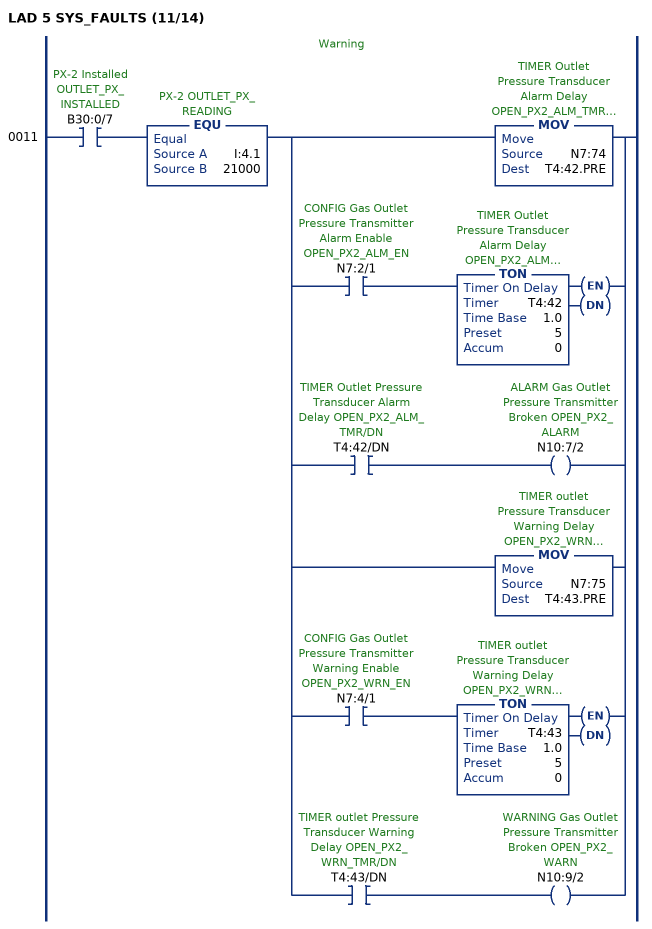
% Rung: 11 %
% Warning %
SOR XIC B30:0/7 EQU I:4.1 21000 BST MOV N7:74 T4:42.PRE NXB XIC N7:2/1 TON T4:42 1.0 5 0 NXB XIC T4:42/DN OTE N10:7/2 NXB MOV N7:75 T4:43.PRE NXB XIC N7:4/1 TON T4:43 1.0 5 0 NXB XIC T4:43/DN OTE N10:9/2 BND EOR
%   B30:0/7  OUTLET_PX_INSTALLED  "PX-2 Installed" %
%   I:4.1  OUTLET_PX_READING  "PX-2" %
%   N7:74  OPEN_PX2_ALM_DLY  "CONFIG Gas Outlet Pressure Transducer Alarm Delay" %
%   T4:42  OPEN_PX2_ALM_TMR  "TIMER Outlet Pressure Transducer Alarm Delay" %
%   N7:2/1  OPEN_PX2_ALM_EN  "CONFIG Gas Outlet Pressure Transmitter Alarm Enable" %
%   N10:7/2  OPEN_PX2_ALARM  "ALARM Gas Outlet Pressure Transmitter Broken" %
%   N7:75  OPEN_PX2_WRN_DLY  "CONFIG Gas Outlet Pressure Transducer Warning Delay" %
%   T4:43  OPEN_PX2_WRN_TMR  "TIMER outlet Pressure Transducer Warning Delay" %
%   N7:4/1  OPEN_PX2_WRN_EN  "CONFIG Gas Outlet Pressure Transmitter Warning Enable" %
%   N10:9/2  OPEN_PX2_WARN  "WARNING Gas Outlet Pressure Transmitter Broken" %

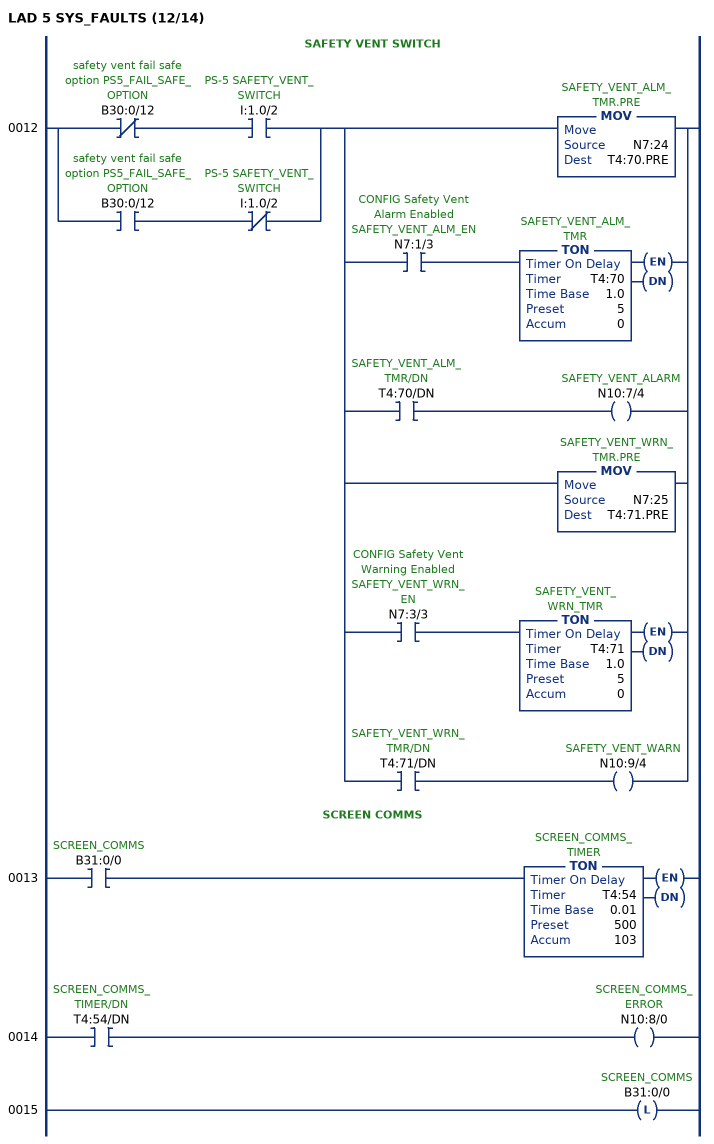
% Rung: 12 %
% TITLE: SAFETY VENT SWITCH %
SOR BST XIO B30:0/12 XIC I:1.0/2 NXB XIC B30:0/12 XIO I:1.0/2 BND BST MOV N7:24 T4:70.PRE NXB XIC N7:1/3 TON T4:70 1.0 5 0 NXB XIC T4:70/DN OTE N10:7/4 NXB MOV N7:25 T4:71.PRE NXB XIC N7:3/3 TON T4:71 1.0 5 0 NXB XIC T4:71/DN OTE N10:9/4 BND EOR
%   B30:0/12  PS5_FAIL_SAFE_OPTION  "safety vent fail safe option" %
%   I:1.0/2  SAFETY_VENT_SWITCH  "PS-5" %
%   N7:24  SAFETY_VENT_ALM_DLY  "CONFIG Safety Vent Alarm Delay" %
%   T4:70  SAFETY_VENT_ALM_TMR %
%   N7:1/3  SAFETY_VENT_ALM_EN  "CONFIG Safety Vent Alarm Enabled" %
%   N10:7/4  SAFETY_VENT_ALARM %
%   N7:25  SAFETY_VENT_WRN_DLY  "CONFIG Safety Vent Warning Delay" %
%   T4:71  SAFETY_VENT_WRN_TMR %
%   N7:3/3  SAFETY_VENT_WRN_EN  "CONFIG Safety Vent Warning Enabled" %
%   N10:9/4  SAFETY_VENT_WARN %
% Rung: 13 %
% TITLE: SCREEN COMMS %
SOR XIC B31:0/0 TON T4:54 0.01 500 103 EOR
%   B31:0/0  SCREEN_COMMS %
%   T4:54  SCREEN_COMMS_TIMER %
% Rung: 14 %
SOR XIC T4:54/DN OTE N10:8/0 EOR
%   T4:54  SCREEN_COMMS_TIMER %
%   N10:8/0  SCREEN_COMMS_ERROR %
% Rung: 15 %
SOR OTL B31:0/0 EOR
%   B31:0/0  SCREEN_COMMS %

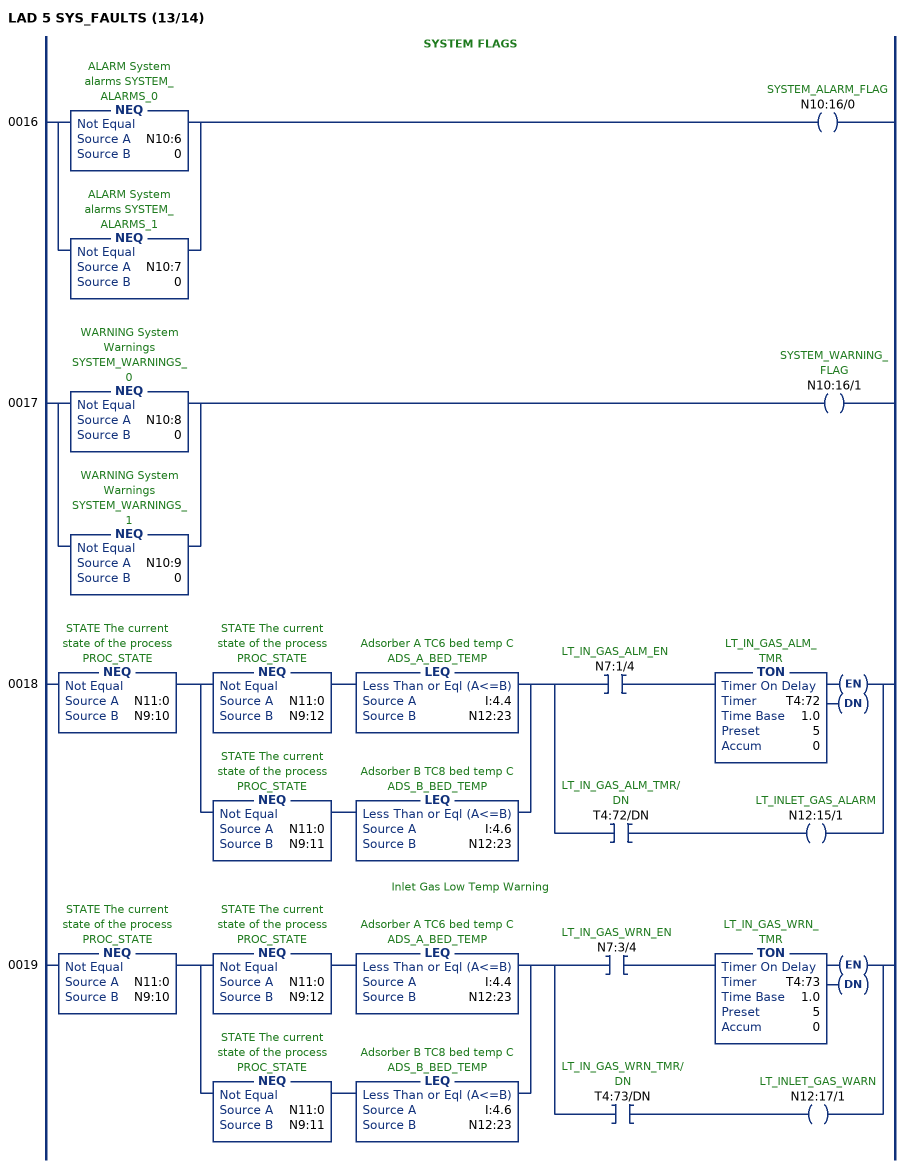
% Rung: 16 %
% TITLE: SYSTEM FLAGS %
SOR BST NEQ N10:6 0 NXB NEQ N10:7 0 BND OTE N10:16/0 EOR
%   N10:6  SYSTEM_ALARMS_0  "ALARM System alarms" %
%   N10:7  SYSTEM_ALARMS_1  "ALARM System alarms" %
%   N10:16/0  SYSTEM_ALARM_FLAG %
% Rung: 17 %
SOR BST NEQ N10:8 0 NXB NEQ N10:9 0 BND OTE N10:16/1 EOR
%   N10:8  SYSTEM_WARNINGS_0  "WARNING System Warnings" %
%   N10:9  SYSTEM_WARNINGS_1  "WARNING System Warnings" %
%   N10:16/1  SYSTEM_WARNING_FLAG %
% Rung: 18 %
SOR NEQ N11:0 N9:10 BST NEQ N11:0 N9:12 LEQ I:4.4 N12:23 NXB NEQ N11:0 N9:11 LEQ I:4.6 N12:23 BND BST XIC N7:1/4 TON T4:72 1.0 5 0 NXB XIC T4:72/DN OTE N12:15/1 BND EOR
%   N11:0  PROC_STATE  "STATE The current state of the process" %
%   N9:10  PROCESS_STANDBY %
%   N9:12  PROC_REGEN_A  "STATE Process Purify B" %
%   I:4.4  ADS_A_BED_TEMP  "Adsorber A TC6 bed temp C" %
%   N12:23  LT_INLET_GAS_ALM_SP %
%   N9:11  PROC_REGEN_B  "STATE Process Purify A" %
%   I:4.6  ADS_B_BED_TEMP  "Adsorber B TC8 bed temp C" %
%   N7:1/4  LT_IN_GAS_ALM_EN %
%   T4:72  LT_IN_GAS_ALM_TMR %
%   N12:15/1  LT_INLET_GAS_ALARM %
% Rung: 19 %
% Inlet Gas Low Temp Warning %
SOR NEQ N11:0 N9:10 BST NEQ N11:0 N9:12 LEQ I:4.4 N12:23 NXB NEQ N11:0 N9:11 LEQ I:4.6 N12:23 BND BST XIC N7:3/4 TON T4:73 1.0 5 0 NXB XIC T4:73/DN OTE N12:17/1 BND EOR
%   N11:0  PROC_STATE  "STATE The current state of the process" %
%   N9:10  PROCESS_STANDBY %
%   N9:12  PROC_REGEN_A  "STATE Process Purify B" %
%   I:4.4  ADS_A_BED_TEMP  "Adsorber A TC6 bed temp C" %
%   N12:23  LT_INLET_GAS_ALM_SP %
%   N9:11  PROC_REGEN_B  "STATE Process Purify A" %
%   I:4.6  ADS_B_BED_TEMP  "Adsorber B TC8 bed temp C" %
%   N7:3/4  LT_IN_GAS_WRN_EN %
%   T4:73  LT_IN_GAS_WRN_TMR %
%   N12:17/1  LT_INLET_GAS_WARN %

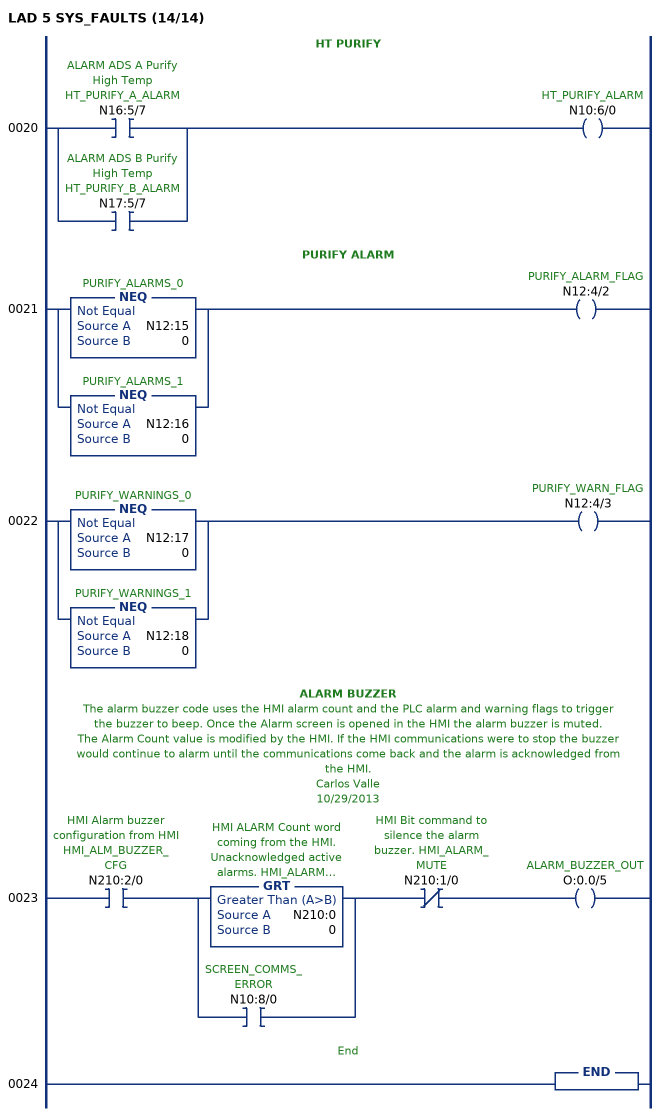
% Rung: 20 %
% TITLE: HT PURIFY %
SOR BST XIC N16:5/7 NXB XIC N17:5/7 BND OTE N10:6/0 EOR
%   N16:5/7  HT_PURIFY_A_ALARM  "ALARM ADS A Purify High Temp" %
%   N17:5/7  HT_PURIFY_B_ALARM  "ALARM ADS B Purify High Temp" %
%   N10:6/0  HT_PURIFY_ALARM %
% Rung: 21 %
% TITLE: PURIFY ALARM %
SOR BST NEQ N12:15 0 NXB NEQ N12:16 0 BND OTE N12:4/2 EOR
%   N12:15  PURIFY_ALARMS_0 %
%   N12:16  PURIFY_ALARMS_1 %
%   N12:4/2  PURIFY_ALARM_FLAG %
% Rung: 22 %
SOR BST NEQ N12:17 0 NXB NEQ N12:18 0 BND OTE N12:4/3 EOR
%   N12:17  PURIFY_WARNINGS_0 %
%   N12:18  PURIFY_WARNINGS_1 %
%   N12:4/3  PURIFY_WARN_FLAG %
% Rung: 23 %
% TITLE: ALARM BUZZER %
% The alarm buzzer code uses the HMI alarm count and the PLC alarm and warning flags to trigger the buzzer to beep. Once the Alarm screen is opened in the HMI the alarm buzzer is muted.
% The Alarm Count value is modified by the HMI. If the HMI communications were to stop the buzzer would continue to alarm until the communications come back and the alarm is acknowledged from the HMI.
% Carlos Valle
% 10/29/2013 %
SOR XIC N210:2/0 BST GRT N210:0 0 NXB XIC N10:8/0 BND XIO N210:1/0 OTE O:0.0/5 EOR
%   N210:2/0  HMI_ALM_BUZZER_CFG  "HMI Alarm buzzer configuration from HMI" %
%   N210:0  HMI_ALARM_COUNT  "HMI ALARM Count word coming from the HMI. Unacknowledged active alarms." %
%   N10:8/0  SCREEN_COMMS_ERROR %
%   N210:1/0  HMI_ALARM_MUTE  "HMI Bit command to silence the alarm buzzer." %
%   O:0.0/5  ALARM_BUZZER_OUT %
% Rung: 24 %
% End %
SOR END EOR

LADDER 6 "SYSTEM"    % Controls the system %
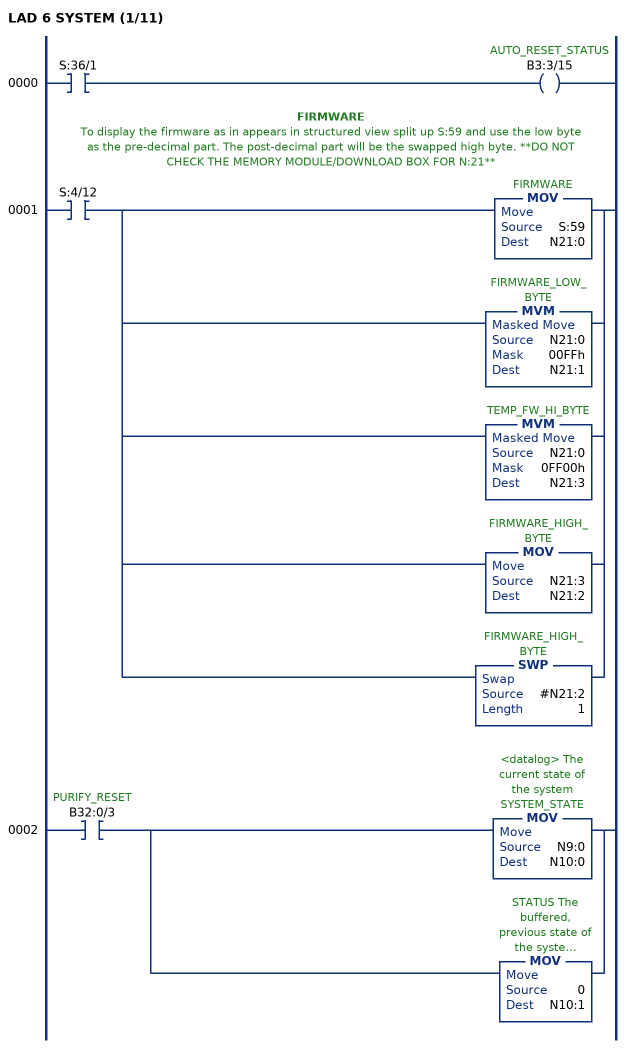
% Rung: 0 %
SOR XIC S:36/1 OTE B3:3/15 EOR
%   B3:3/15  AUTO_RESET_STATUS %
% Rung: 1 %
% TITLE: FIRMWARE %
% To display the firmware as in appears in structured view split up S:59 and use the low byte as the pre-decimal part. The post-decimal part will be the swapped high byte. **DO NOT CHECK THE MEMORY MODULE/DOWNLOAD BOX FOR N:21** %
SOR XIC S:4/12 BST MOV S:59 N21:0 NXB MVM N21:0 00FFh N21:1 NXB MVM N21:0 0FF00h N21:3 NXB MOV N21:3 N21:2 NXB SWP #N21:2 1 BND EOR
%   S:59  "Operating System FRN" %
%   N21:0  FIRMWARE %
%   N21:1  FIRMWARE_LOW_BYTE %
%   N21:3  TEMP_FW_HI_BYTE %
%   N21:2  FIRMWARE_HIGH_BYTE %
% Rung: 2 %
SOR XIC B32:0/3 BST MOV N9:0 N10:0 NXB MOV 0 N10:1 BND EOR
%   B32:0/3  PURIFY_RESET %
%   N9:0  SYSTEM_STANDBY  "STATE System Standby" %
%   N10:0  SYSTEM_STATE  "<datalog> The current state of the system" %
%   N10:1  SYSTEM_BUFFER  "STATUS The buffered, previous state of the system" %

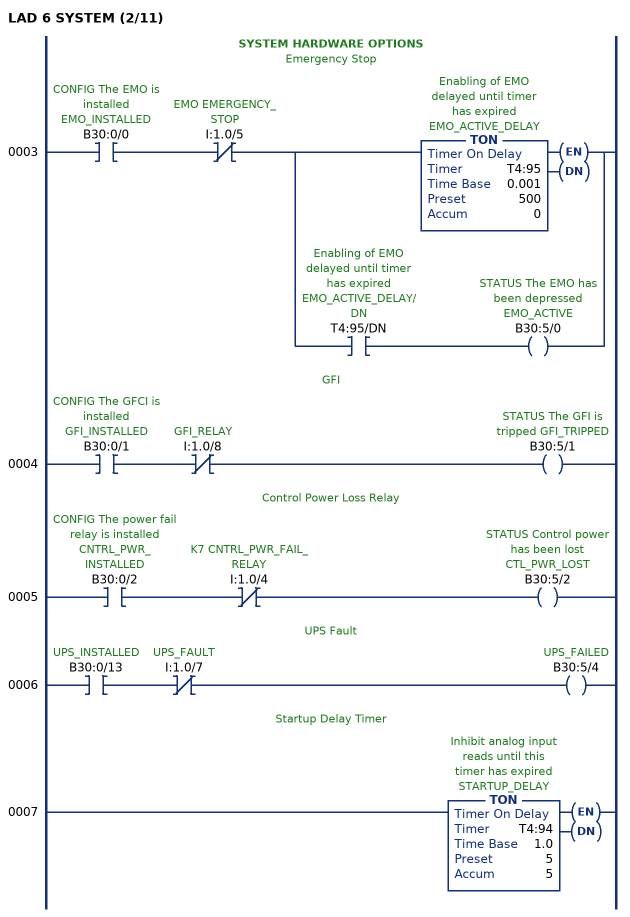
% Rung: 3 %
% TITLE: SYSTEM HARDWARE OPTIONS %
% Emergency Stop %
SOR XIC B30:0/0 XIO I:1.0/5 BST TON T4:95 0.001 500 0 NXB XIC T4:95/DN OTE B30:5/0 BND EOR
%   B30:0/0  EMO_INSTALLED  "CONFIG The EMO is installed" %
%   I:1.0/5  EMERGENCY_STOP  "EMO" %
%   T4:95  EMO_ACTIVE_DELAY  "Enabling of EMO delayed until timer has expired" %
%   B30:5/0  EMO_ACTIVE  "STATUS The EMO has been depressed" %
% Rung: 4 %
% GFI %
SOR XIC B30:0/1 XIO I:1.0/8 OTE B30:5/1 EOR
%   B30:0/1  GFI_INSTALLED  "CONFIG The GFCI is installed" %
%   I:1.0/8  GFI_RELAY %
%   B30:5/1  GFI_TRIPPED  "STATUS The GFI is tripped" %
% Rung: 5 %
% Control Power Loss Relay %
SOR XIC B30:0/2 XIO I:1.0/4 OTE B30:5/2 EOR
%   B30:0/2  CNTRL_PWR_INSTALLED  "CONFIG The power fail relay is installed" %
%   I:1.0/4  CNTRL_PWR_FAIL_RELAY  "K7" %
%   B30:5/2  CTL_PWR_LOST  "STATUS Control power has been lost" %
% Rung: 6 %
% UPS Fault %
SOR XIC B30:0/13 XIO I:1.0/7 OTE B30:5/4 EOR
%   B30:0/13  UPS_INSTALLED %
%   I:1.0/7  UPS_FAULT %
%   B30:5/4  UPS_FAILED %
% Rung: 7 %
% Startup Delay Timer %
SOR TON T4:94 1.0 5 5 EOR
%   T4:94  STARTUP_DELAY  "Inhibit analog input reads until this timer has expired" %

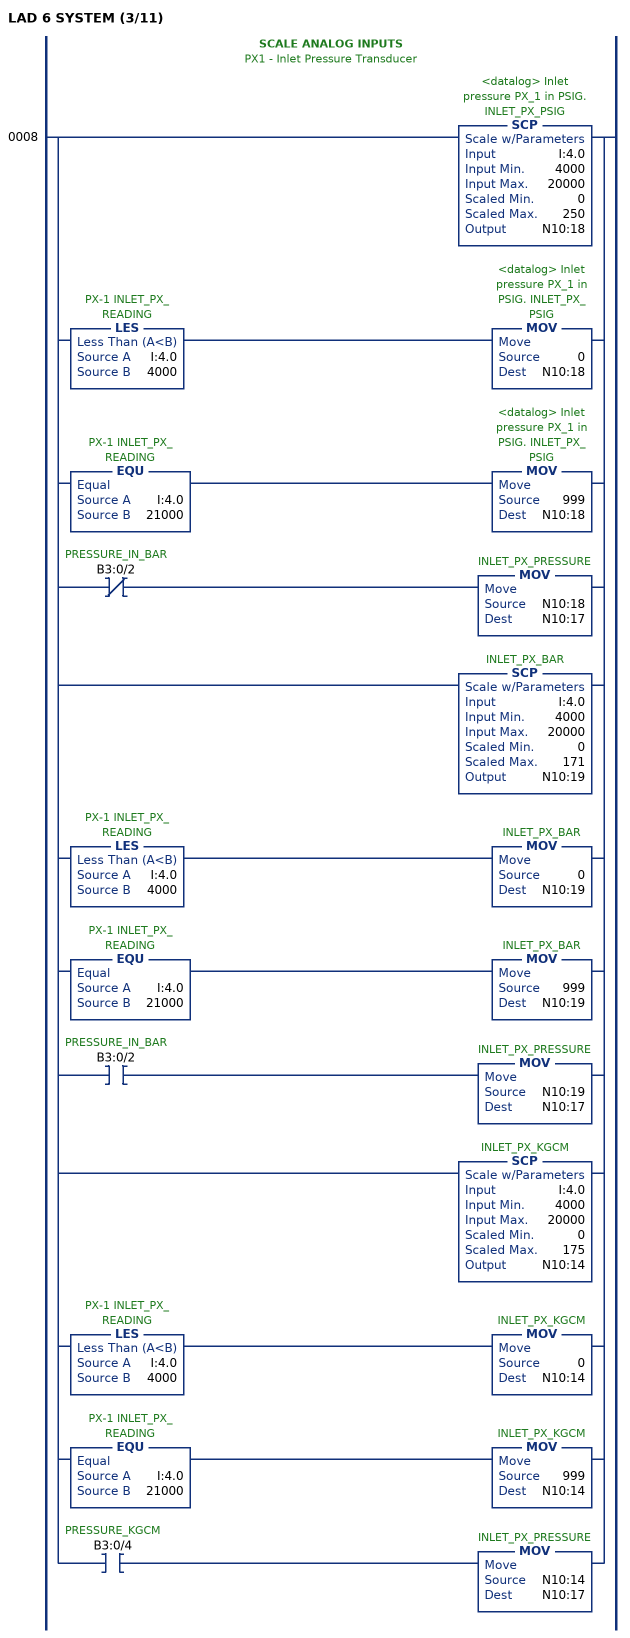
% Rung: 8 %
% TITLE: SCALE ANALOG INPUTS %
% PX1 - Inlet Pressure Transducer %
SOR BST SCP I:4.0 4000 20000 0 250 N10:18 NXB LES I:4.0 4000 MOV 0 N10:18 NXB EQU I:4.0 21000 MOV 999 N10:18 NXB XIO B3:0/2 MOV N10:18 N10:17 NXB SCP I:4.0 4000 20000 0 171 N10:19 NXB LES I:4.0 4000 MOV 0 N10:19 NXB EQU I:4.0 21000 MOV 999 N10:19 NXB XIC B3:0/2 MOV N10:19 N10:17 NXB SCP I:4.0 4000 20000 0 175 N10:14 NXB LES I:4.0 4000 MOV 0 N10:14 NXB EQU I:4.0 21000 MOV 999 N10:14 NXB XIC B3:0/4 MOV N10:14 N10:17 BND EOR
%   I:4.0  INLET_PX_READING  "PX-1" %
%   N10:18  INLET_PX_PSIG  "<datalog> Inlet pressure PX_1 in PSIG." %
%   B3:0/2  PRESSURE_IN_BAR %
%   N10:17  INLET_PX_PRESSURE %
%   N10:19  INLET_PX_BAR %
%   N10:14  INLET_PX_KGCM %
%   B3:0/4  PRESSURE_KGCM %

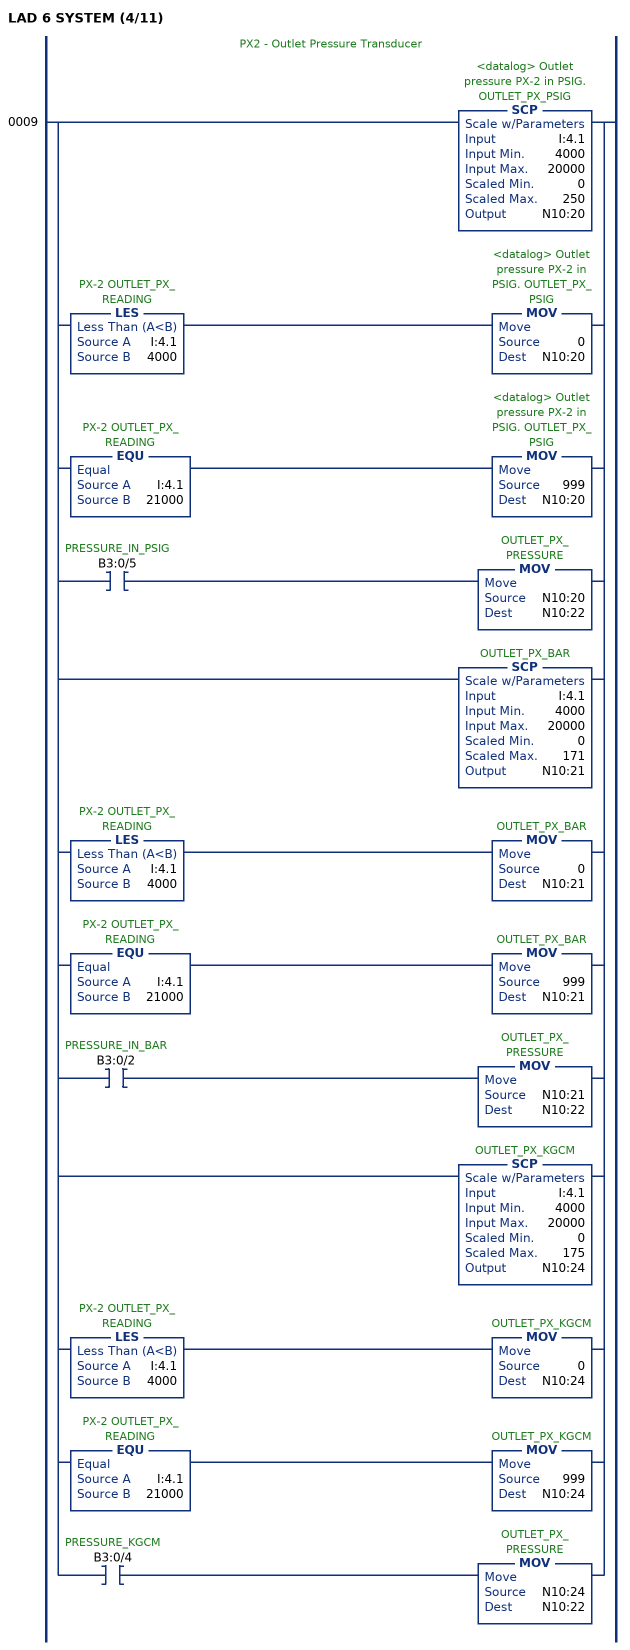
% Rung: 9 %
% PX2 - Outlet Pressure Transducer %
SOR BST SCP I:4.1 4000 20000 0 250 N10:20 NXB LES I:4.1 4000 MOV 0 N10:20 NXB EQU I:4.1 21000 MOV 999 N10:20 NXB XIC B3:0/5 MOV N10:20 N10:22 NXB SCP I:4.1 4000 20000 0 171 N10:21 NXB LES I:4.1 4000 MOV 0 N10:21 NXB EQU I:4.1 21000 MOV 999 N10:21 NXB XIC B3:0/2 MOV N10:21 N10:22 NXB SCP I:4.1 4000 20000 0 175 N10:24 NXB LES I:4.1 4000 MOV 0 N10:24 NXB EQU I:4.1 21000 MOV 999 N10:24 NXB XIC B3:0/4 MOV N10:24 N10:22 BND EOR
%   I:4.1  OUTLET_PX_READING  "PX-2" %
%   N10:20  OUTLET_PX_PSIG  "<datalog> Outlet pressure PX-2 in PSIG." %
%   B3:0/5  PRESSURE_IN_PSIG %
%   N10:22  OUTLET_PX_PRESSURE %
%   N10:21  OUTLET_PX_BAR %
%   B3:0/2  PRESSURE_IN_BAR %
%   N10:24  OUTLET_PX_KGCM %
%   B3:0/4  PRESSURE_KGCM %

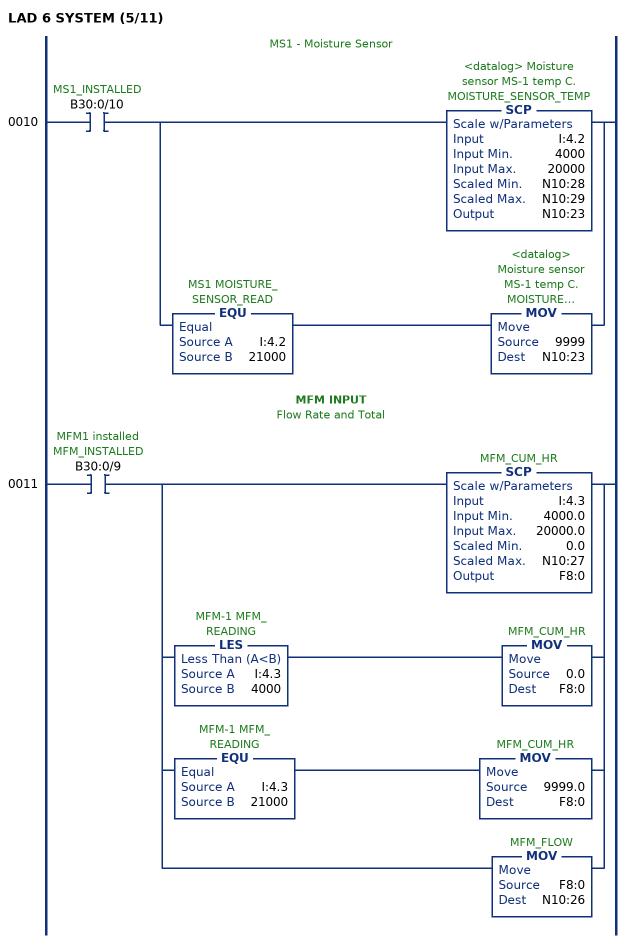
% Rung: 10 %
% MS1 - Moisture Sensor %
SOR XIC B30:0/10 BST SCP I:4.2 4000 20000 N10:28 N10:29 N10:23 NXB EQU I:4.2 21000 MOV 9999 N10:23 BND EOR
%   B30:0/10  MS1_INSTALLED %
%   I:4.2  MOISTURE_SENSOR_READ  "MS1" %
%   N10:28  H20_SENS_MIN %
%   N10:29  H20_SENS_MAX %
%   N10:23  MOISTURE_SENSOR_TEMP  "<datalog> Moisture sensor MS-1 temp C." %
% Rung: 11 %
% TITLE: MFM INPUT %
% Flow Rate and Total %
SOR XIC B30:0/9 BST SCP I:4.3 4000.0 20000.0 0.0 N10:27 F8:0 NXB LES I:4.3 4000 MOV 0.0 F8:0 NXB EQU I:4.3 21000 MOV 9999.0 F8:0 NXB MOV F8:0 N10:26 BND EOR
%   B30:0/9  MFM_INSTALLED  "MFM1 installed" %
%   I:4.3  MFM_READING  "MFM-1" %
%   N10:27  MFM_SCALING %
%   F8:0  MFM_CUM_HR %
%   N10:26  MFM_FLOW %

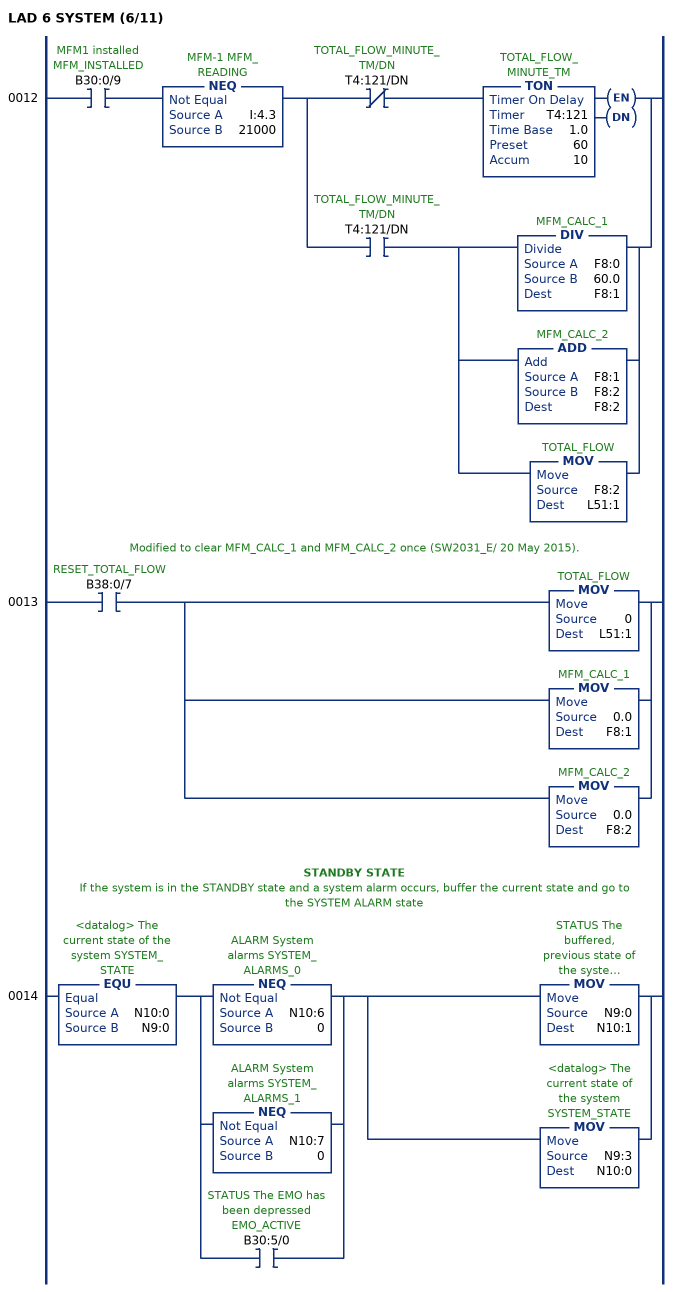
% Rung: 12 %
SOR XIC B30:0/9 NEQ I:4.3 21000 BST XIO T4:121/DN TON T4:121 1.0 60 10 NXB XIC T4:121/DN BST DIV F8:0 60.0 F8:1 NXB ADD F8:1 F8:2 F8:2 NXB MOV F8:2 L51:1 BND BND EOR
%   B30:0/9  MFM_INSTALLED  "MFM1 installed" %
%   I:4.3  MFM_READING  "MFM-1" %
%   T4:121  TOTAL_FLOW_MINUTE_TM %
%   F8:0  MFM_CUM_HR %
%   F8:1  MFM_CALC_1 %
%   F8:2  MFM_CALC_2 %
%   L51:1  TOTAL_FLOW %
% Rung: 13 %
% Modified to clear MFM_CALC_1 and MFM_CALC_2 once (SW2031_E/ 20 May 2015). %
SOR XIC B38:0/7 BST MOV 0 L51:1 NXB MOV 0.0 F8:1 NXB MOV 0.0 F8:2 BND EOR
%   B38:0/7  RESET_TOTAL_FLOW %
%   L51:1  TOTAL_FLOW %
%   F8:1  MFM_CALC_1 %
%   F8:2  MFM_CALC_2 %
% Rung: 14 %
% TITLE: STANDBY STATE %
% If the system is in the STANDBY state and a system alarm occurs, buffer the current state and go to the SYSTEM ALARM state %
SOR EQU N10:0 N9:0 BST NEQ N10:6 0 NXB NEQ N10:7 0 NXB XIC B30:5/0 BND BST MOV N9:0 N10:1 NXB MOV N9:3 N10:0 BND EOR
%   N10:0  SYSTEM_STATE  "<datalog> The current state of the system" %
%   N9:0  SYSTEM_STANDBY  "STATE System Standby" %
%   N10:6  SYSTEM_ALARMS_0  "ALARM System alarms" %
%   N10:7  SYSTEM_ALARMS_1  "ALARM System alarms" %
%   B30:5/0  EMO_ACTIVE  "STATUS The EMO has been depressed" %
%   N10:1  SYSTEM_BUFFER  "STATUS The buffered, previous state of the system" %
%   N9:3  SYSTEM_ALARM  "STATE System Alarm" %

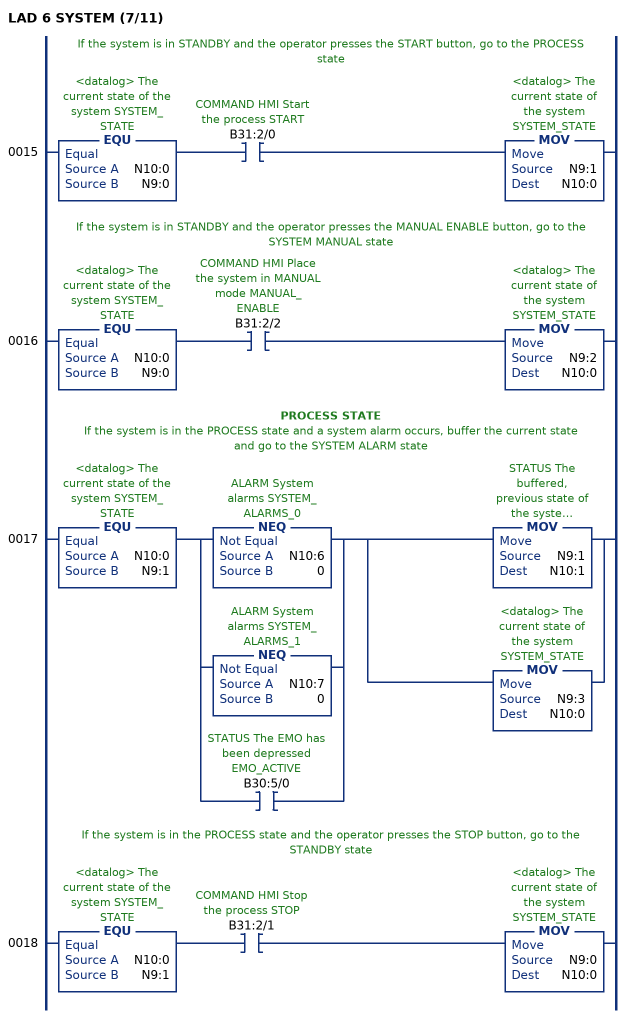
% Rung: 15 %
% If the system is in STANDBY and the operator presses the START button, go to the PROCESS state %
SOR EQU N10:0 N9:0 XIC B31:2/0 MOV N9:1 N10:0 EOR
%   N10:0  SYSTEM_STATE  "<datalog> The current state of the system" %
%   N9:0  SYSTEM_STANDBY  "STATE System Standby" %
%   B31:2/0  START  "COMMAND HMI Start the process" %
%   N9:1  SYSTEM_PROCESS  "STATE System Process" %
% Rung: 16 %
% If the system is in STANDBY and the operator presses the MANUAL ENABLE button, go to the SYSTEM MANUAL state %
SOR EQU N10:0 N9:0 XIC B31:2/2 MOV N9:2 N10:0 EOR
%   N10:0  SYSTEM_STATE  "<datalog> The current state of the system" %
%   N9:0  SYSTEM_STANDBY  "STATE System Standby" %
%   B31:2/2  MANUAL_ENABLE  "COMMAND HMI Place the system in MANUAL mode" %
%   N9:2  SYSTEM_MANUAL  "STATE System Manual" %
% Rung: 17 %
% TITLE: PROCESS STATE %
% If the system is in the PROCESS state and a system alarm occurs, buffer the current state and go to the SYSTEM ALARM state %
SOR EQU N10:0 N9:1 BST NEQ N10:6 0 NXB NEQ N10:7 0 NXB XIC B30:5/0 BND BST MOV N9:1 N10:1 NXB MOV N9:3 N10:0 BND EOR
%   N10:0  SYSTEM_STATE  "<datalog> The current state of the system" %
%   N9:1  SYSTEM_PROCESS  "STATE System Process" %
%   N10:6  SYSTEM_ALARMS_0  "ALARM System alarms" %
%   N10:7  SYSTEM_ALARMS_1  "ALARM System alarms" %
%   B30:5/0  EMO_ACTIVE  "STATUS The EMO has been depressed" %
%   N10:1  SYSTEM_BUFFER  "STATUS The buffered, previous state of the system" %
%   N9:3  SYSTEM_ALARM  "STATE System Alarm" %
% Rung: 18 %
% If the system is in the PROCESS state and the operator presses the STOP button, go to the STANDBY state %
SOR EQU N10:0 N9:1 XIC B31:2/1 MOV N9:0 N10:0 EOR
%   N10:0  SYSTEM_STATE  "<datalog> The current state of the system" %
%   N9:1  SYSTEM_PROCESS  "STATE System Process" %
%   B31:2/1  STOP  "COMMAND HMI Stop the process" %
%   N9:0  SYSTEM_STANDBY  "STATE System Standby" %

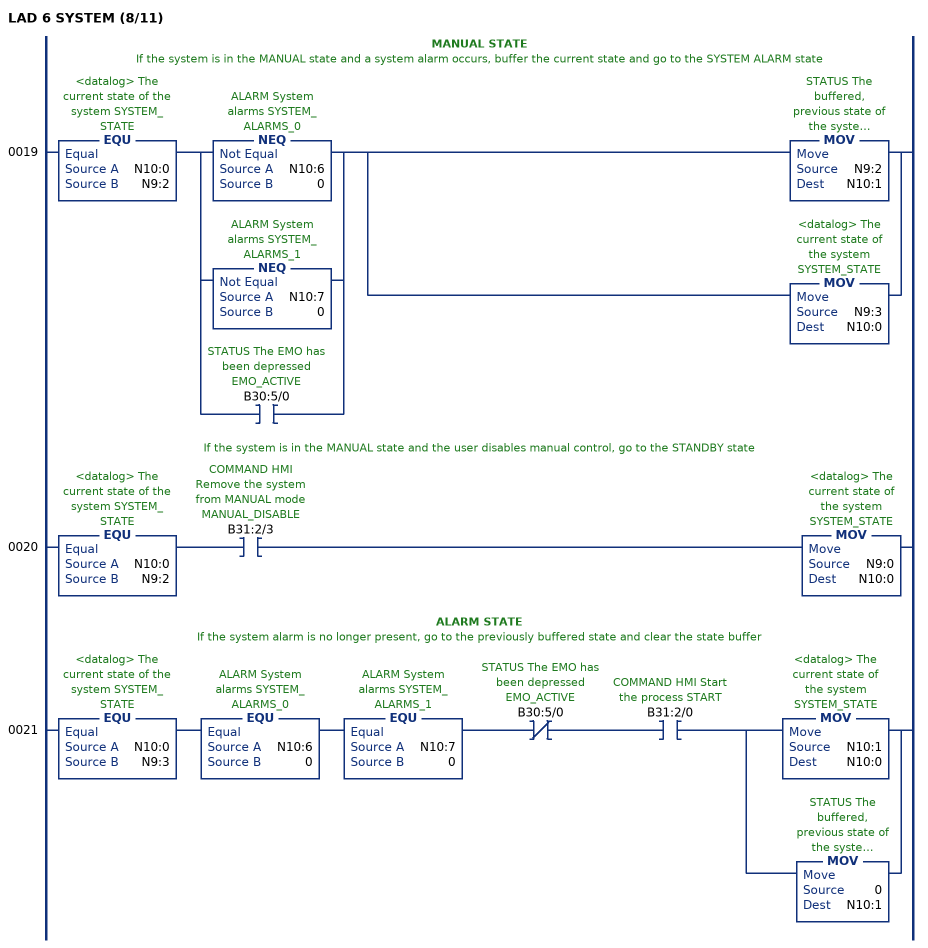
% Rung: 19 %
% TITLE: MANUAL STATE %
% If the system is in the MANUAL state and a system alarm occurs, buffer the current state and go to the SYSTEM ALARM state %
SOR EQU N10:0 N9:2 BST NEQ N10:6 0 NXB NEQ N10:7 0 NXB XIC B30:5/0 BND BST MOV N9:2 N10:1 NXB MOV N9:3 N10:0 BND EOR
%   N10:0  SYSTEM_STATE  "<datalog> The current state of the system" %
%   N9:2  SYSTEM_MANUAL  "STATE System Manual" %
%   N10:6  SYSTEM_ALARMS_0  "ALARM System alarms" %
%   N10:7  SYSTEM_ALARMS_1  "ALARM System alarms" %
%   B30:5/0  EMO_ACTIVE  "STATUS The EMO has been depressed" %
%   N10:1  SYSTEM_BUFFER  "STATUS The buffered, previous state of the system" %
%   N9:3  SYSTEM_ALARM  "STATE System Alarm" %
% Rung: 20 %
% If the system is in the MANUAL state and the user disables manual control, go to the STANDBY state %
SOR EQU N10:0 N9:2 XIC B31:2/3 MOV N9:0 N10:0 EOR
%   N10:0  SYSTEM_STATE  "<datalog> The current state of the system" %
%   N9:2  SYSTEM_MANUAL  "STATE System Manual" %
%   B31:2/3  MANUAL_DISABLE  "COMMAND HMI Remove the system from MANUAL mode" %
%   N9:0  SYSTEM_STANDBY  "STATE System Standby" %
% Rung: 21 %
% TITLE: ALARM STATE %
% If the system alarm is no longer present, go to the previously buffered state and clear the state buffer %
SOR EQU N10:0 N9:3 EQU N10:6 0 EQU N10:7 0 XIO B30:5/0 XIC B31:2/0 BST MOV N10:1 N10:0 NXB MOV 0 N10:1 BND EOR
%   N10:0  SYSTEM_STATE  "<datalog> The current state of the system" %
%   N9:3  SYSTEM_ALARM  "STATE System Alarm" %
%   N10:6  SYSTEM_ALARMS_0  "ALARM System alarms" %
%   N10:7  SYSTEM_ALARMS_1  "ALARM System alarms" %
%   B30:5/0  EMO_ACTIVE  "STATUS The EMO has been depressed" %
%   B31:2/0  START  "COMMAND HMI Start the process" %
%   N10:1  SYSTEM_BUFFER  "STATUS The buffered, previous state of the system" %

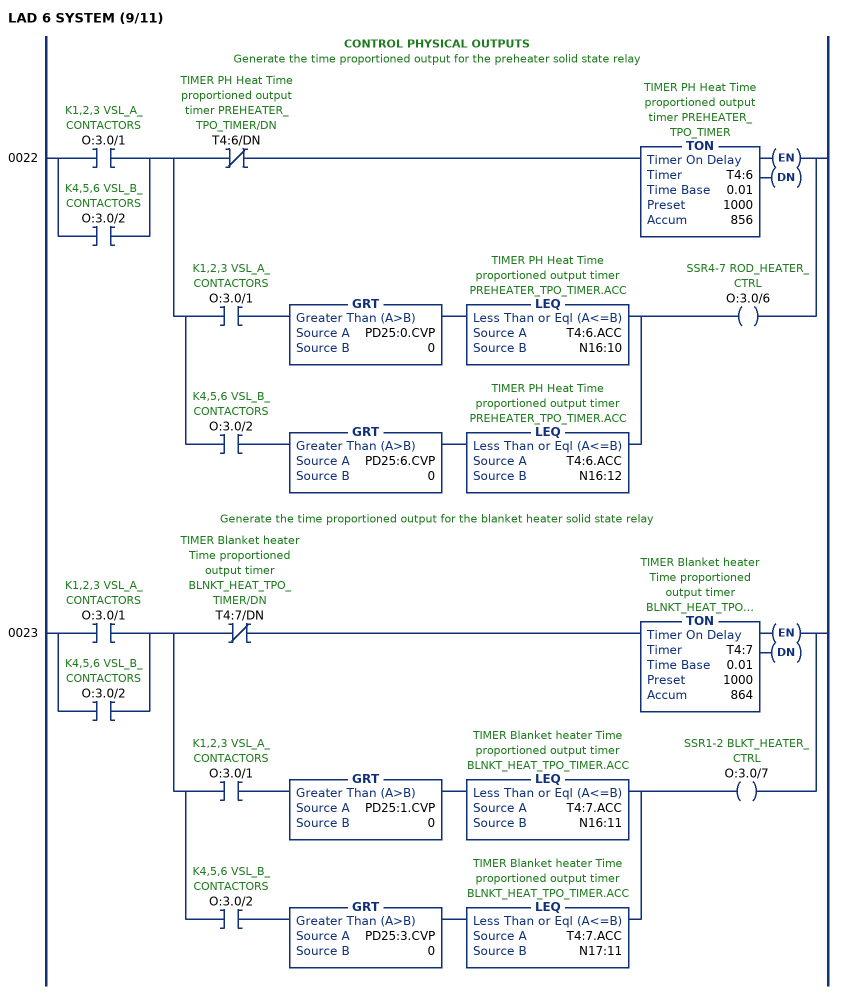
% Rung: 22 %
% TITLE: CONTROL PHYSICAL OUTPUTS %
% Generate the time proportioned output for the preheater solid state relay %
SOR BST XIC O:3.0/1 NXB XIC O:3.0/2 BND BST XIO T4:6/DN TON T4:6 0.01 1000 856 NXB BST XIC O:3.0/1 GRT PD25:0.CVP 0 LEQ T4:6.ACC N16:10 NXB XIC O:3.0/2 GRT PD25:6.CVP 0 LEQ T4:6.ACC N16:12 BND OTE O:3.0/6 BND EOR
%   O:3.0/1  VSL_A_CONTACTORS  "K1,2,3" %
%   O:3.0/2  VSL_B_CONTACTORS  "K4,5,6" %
%   T4:6  PREHEATER_TPO_TIMER  "TIMER PH Heat Time proportioned output timer" %
%   N16:10  ADS_A_PH_OUTPUT  "<datalog> Adsorber A heater duty cycle %" %
%   N16:12  ADS_B_PH_OUTPUT  "<datalog> Adsorber B heater duty cycle %" %
%   O:3.0/6  ROD_HEATER_CTRL  "SSR4-7" %
% Rung: 23 %
% Generate the time proportioned output for the blanket heater solid state relay %
SOR BST XIC O:3.0/1 NXB XIC O:3.0/2 BND BST XIO T4:7/DN TON T4:7 0.01 1000 864 NXB BST XIC O:3.0/1 GRT PD25:1.CVP 0 LEQ T4:7.ACC N16:11 NXB XIC O:3.0/2 GRT PD25:3.CVP 0 LEQ T4:7.ACC N17:11 BND OTE O:3.0/7 BND EOR
%   O:3.0/1  VSL_A_CONTACTORS  "K1,2,3" %
%   O:3.0/2  VSL_B_CONTACTORS  "K4,5,6" %
%   T4:7  BLNKT_HEAT_TPO_TIMER  "TIMER Blanket heater Time proportioned output timer" %
%   N16:11  ADS_A_BLNKT_OUTPUT  "CONTROL ADS A Blanket output (percent)" %
%   N17:11  ADS_B_BLNKT_OUTPUT  "CONTROL ADS A Blanket output" %
%   O:3.0/7  BLKT_HEATER_CTRL  "SSR1-2" %

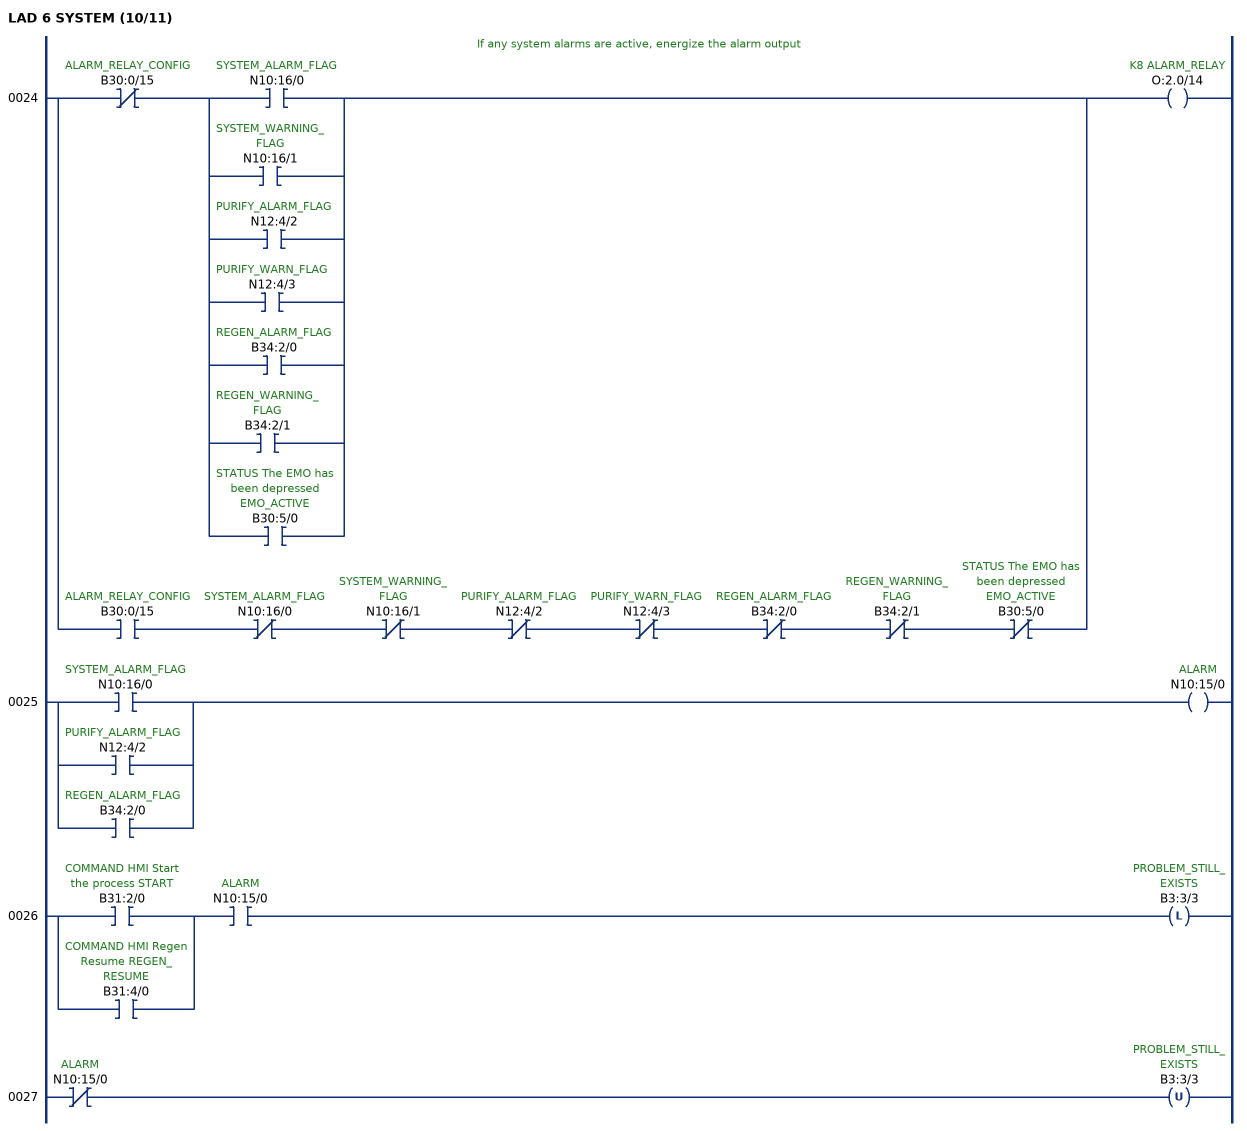
% Rung: 24 %
% If any system alarms are active, energize the alarm output %
SOR BST XIO B30:0/15 BST XIC N10:16/0 NXB XIC N10:16/1 NXB XIC N12:4/2 NXB XIC N12:4/3 NXB XIC B34:2/0 NXB XIC B34:2/1 NXB XIC B30:5/0 BND NXB XIC B30:0/15 XIO N10:16/0 XIO N10:16/1 XIO N12:4/2 XIO N12:4/3 XIO B34:2/0 XIO B34:2/1 XIO B30:5/0 BND OTE O:2.0/14 EOR
%   B30:0/15  ALARM_RELAY_CONFIG %
%   N10:16/0  SYSTEM_ALARM_FLAG %
%   N10:16/1  SYSTEM_WARNING_FLAG %
%   N12:4/2  PURIFY_ALARM_FLAG %
%   N12:4/3  PURIFY_WARN_FLAG %
%   B34:2/0  REGEN_ALARM_FLAG %
%   B34:2/1  REGEN_WARNING_FLAG %
%   B30:5/0  EMO_ACTIVE  "STATUS The EMO has been depressed" %
%   O:2.0/14  ALARM_RELAY  "K8" %
% Rung: 25 %
SOR BST XIC N10:16/0 NXB XIC N12:4/2 NXB XIC B34:2/0 BND OTE N10:15/0 EOR
%   N10:16/0  SYSTEM_ALARM_FLAG %
%   N12:4/2  PURIFY_ALARM_FLAG %
%   B34:2/0  REGEN_ALARM_FLAG %
%   N10:15/0  ALARM %
% Rung: 26 %
SOR BST XIC B31:2/0 NXB XIC B31:4/0 BND XIC N10:15/0 OTL B3:3/3 EOR
%   B31:2/0  START  "COMMAND HMI Start the process" %
%   B31:4/0  REGEN_RESUME  "COMMAND HMI Regen Resume" %
%   N10:15/0  ALARM %
%   B3:3/3  PROBLEM_STILL_EXISTS %
% Rung: 27 %
SOR XIO N10:15/0 OTU B3:3/3 EOR
%   N10:15/0  ALARM %
%   B3:3/3  PROBLEM_STILL_EXISTS %

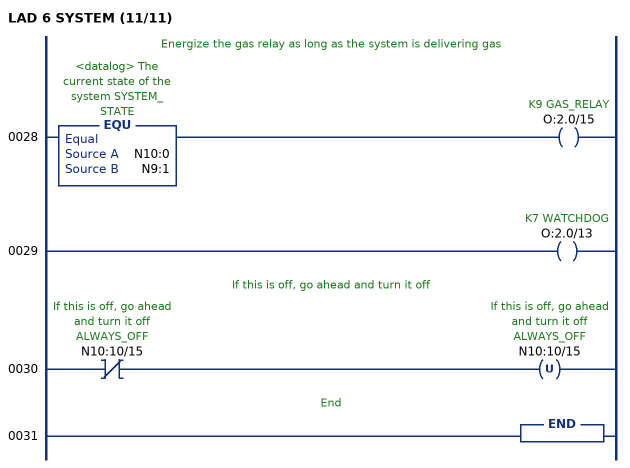
% Rung: 28 %
% Energize the gas relay as long as the system is delivering gas %
SOR EQU N10:0 N9:1 OTE O:2.0/15 EOR
%   N10:0  SYSTEM_STATE  "<datalog> The current state of the system" %
%   N9:1  SYSTEM_PROCESS  "STATE System Process" %
%   O:2.0/15  GAS_RELAY  "K9" %
% Rung: 29 %
SOR OTE O:2.0/13 EOR
%   O:2.0/13  WATCHDOG  "K7" %
% Rung: 30 %
% If this is off, go ahead and turn it off %
SOR XIO N10:10/15 OTU N10:10/15 EOR
%   N10:10/15  ALWAYS_OFF  "If this is off, go ahead and turn it off" %
% Rung: 31 %
% End %
SOR END EOR

LADDER 7 "PROCESSING"    % Runs the processing control %
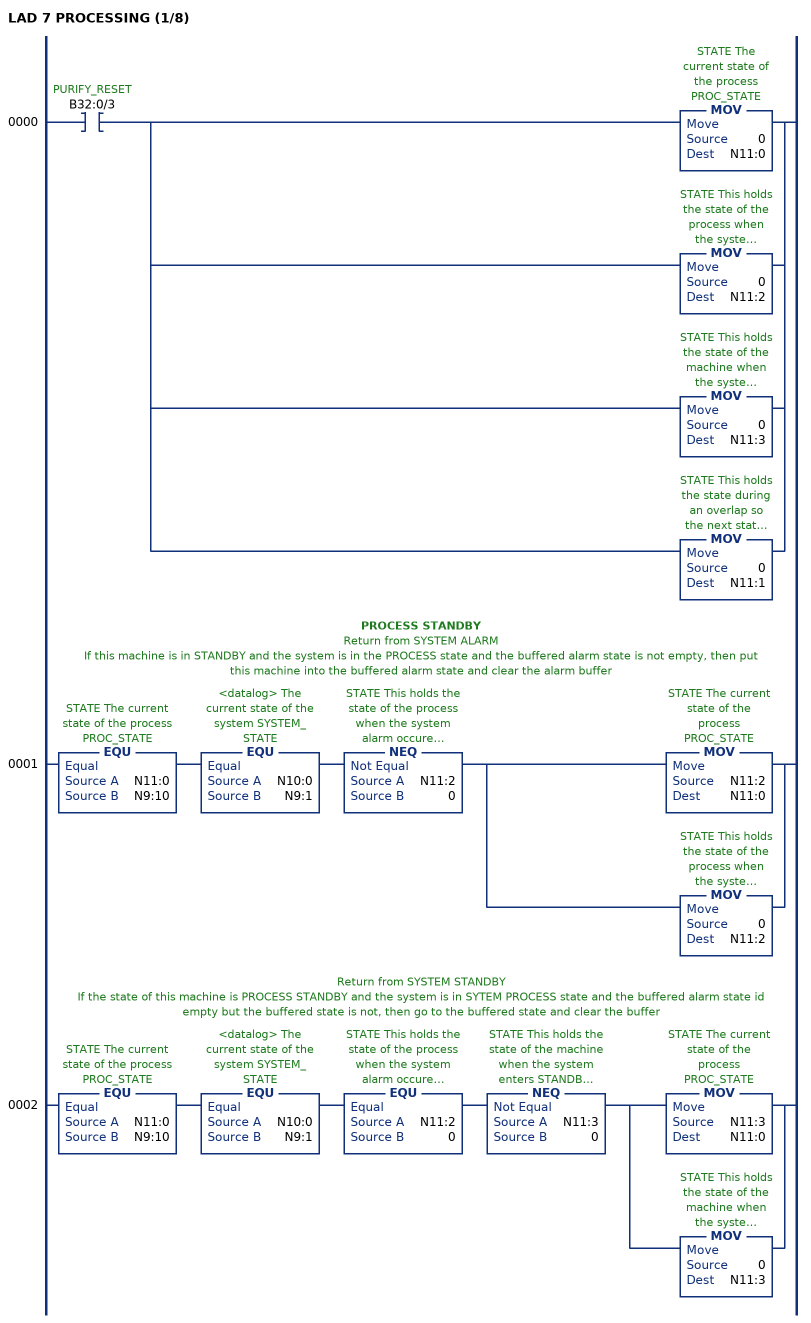
% Rung: 0 %
SOR XIC B32:0/3 BST MOV 0 N11:0 NXB MOV 0 N11:2 NXB MOV 0 N11:3 NXB MOV 0 N11:1 BND EOR
%   B32:0/3  PURIFY_RESET %
%   N11:0  PROC_STATE  "STATE The current state of the process" %
%   N11:2  PROC_ALARM_BUFFER  "STATE This holds the state of the process when the system alarm occured" %
%   N11:3  PROC_STANDBY_BUFFER  "STATE This holds the state of the machine when the system enters STANDBY state" %
%   N11:1  PROC_OVERLAP_BUFFER  "STATE This holds the state during an overlap so the next state can be determined" %
% Rung: 1 %
% TITLE: PROCESS STANDBY %
% Return from SYSTEM ALARM
% If this machine is in STANDBY and the system is in the PROCESS state and the buffered alarm state is not empty, then put this machine into the buffered alarm state and clear the alarm buffer %
SOR EQU N11:0 N9:10 EQU N10:0 N9:1 NEQ N11:2 0 BST MOV N11:2 N11:0 NXB MOV 0 N11:2 BND EOR
%   N11:0  PROC_STATE  "STATE The current state of the process" %
%   N9:10  PROCESS_STANDBY %
%   N10:0  SYSTEM_STATE  "<datalog> The current state of the system" %
%   N9:1  SYSTEM_PROCESS  "STATE System Process" %
%   N11:2  PROC_ALARM_BUFFER  "STATE This holds the state of the process when the system alarm occured" %
% Rung: 2 %
% Return from SYSTEM STANDBY
% If the state of this machine is PROCESS STANDBY and the system is in SYTEM PROCESS state and the buffered alarm state id empty but the buffered state is not, then go to the buffered state and clear the buffer %
SOR EQU N11:0 N9:10 EQU N10:0 N9:1 EQU N11:2 0 NEQ N11:3 0 BST MOV N11:3 N11:0 NXB MOV 0 N11:3 BND EOR
%   N11:0  PROC_STATE  "STATE The current state of the process" %
%   N9:10  PROCESS_STANDBY %
%   N10:0  SYSTEM_STATE  "<datalog> The current state of the system" %
%   N9:1  SYSTEM_PROCESS  "STATE System Process" %
%   N11:2  PROC_ALARM_BUFFER  "STATE This holds the state of the process when the system alarm occured" %
%   N11:3  PROC_STANDBY_BUFFER  "STATE This holds the state of the machine when the system enters STANDBY state" %

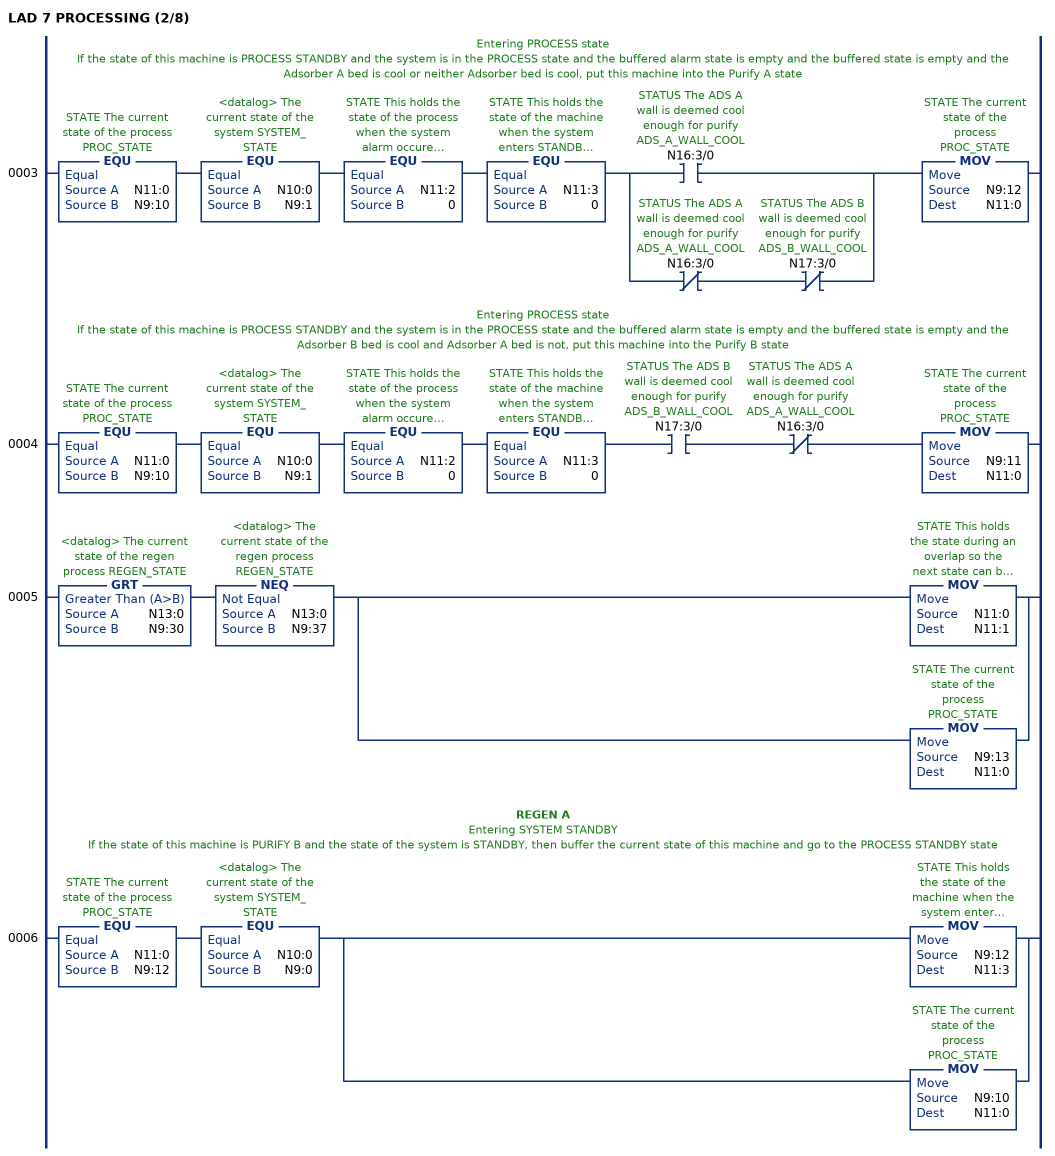
% Rung: 3 %
% Entering PROCESS state
% If the state of this machine is PROCESS STANDBY and the system is in the PROCESS state and the buffered alarm state is empty and the buffered state is empty and the Adsorber A bed is cool or neither Adsorber bed is cool, put this machine into the Purify A state %
SOR EQU N11:0 N9:10 EQU N10:0 N9:1 EQU N11:2 0 EQU N11:3 0 BST XIC N16:3/0 NXB XIO N16:3/0 XIO N17:3/0 BND MOV N9:12 N11:0 EOR
%   N11:0  PROC_STATE  "STATE The current state of the process" %
%   N9:10  PROCESS_STANDBY %
%   N10:0  SYSTEM_STATE  "<datalog> The current state of the system" %
%   N9:1  SYSTEM_PROCESS  "STATE System Process" %
%   N11:2  PROC_ALARM_BUFFER  "STATE This holds the state of the process when the system alarm occured" %
%   N11:3  PROC_STANDBY_BUFFER  "STATE This holds the state of the machine when the system enters STANDBY state" %
%   N16:3/0  ADS_A_WALL_COOL  "STATUS The ADS A wall is deemed cool enough for purify" %
%   N17:3/0  ADS_B_WALL_COOL  "STATUS The ADS B wall is deemed cool enough for purify" %
%   N9:12  PROC_REGEN_A  "STATE Process Purify B" %
% Rung: 4 %
% Entering PROCESS state
% If the state of this machine is PROCESS STANDBY and the system is in the PROCESS state and the buffered alarm state is empty and the buffered state is empty and the Adsorber B bed is cool and Adsorber A bed is not, put this machine into the Purify B state %
SOR EQU N11:0 N9:10 EQU N10:0 N9:1 EQU N11:2 0 EQU N11:3 0 XIC N17:3/0 XIO N16:3/0 MOV N9:11 N11:0 EOR
%   N11:0  PROC_STATE  "STATE The current state of the process" %
%   N9:10  PROCESS_STANDBY %
%   N10:0  SYSTEM_STATE  "<datalog> The current state of the system" %
%   N9:1  SYSTEM_PROCESS  "STATE System Process" %
%   N11:2  PROC_ALARM_BUFFER  "STATE This holds the state of the process when the system alarm occured" %
%   N11:3  PROC_STANDBY_BUFFER  "STATE This holds the state of the machine when the system enters STANDBY state" %
%   N17:3/0  ADS_B_WALL_COOL  "STATUS The ADS B wall is deemed cool enough for purify" %
%   N16:3/0  ADS_A_WALL_COOL  "STATUS The ADS A wall is deemed cool enough for purify" %
%   N9:11  PROC_REGEN_B  "STATE Process Purify A" %
% Rung: 5 %
SOR GRT N13:0 N9:30 NEQ N13:0 N9:37 BST MOV N11:0 N11:1 NXB MOV N9:13 N11:0 BND EOR
%   N13:0  REGEN_STATE  "<datalog> The current state of the regen process" %
%   N9:30  REGEN_STANDBY  "STATE Regen Standby" %
%   N9:37  REGEN_ALARM  "STATE Regen Alarm" %
%   N11:0  PROC_STATE  "STATE The current state of the process" %
%   N11:1  PROC_OVERLAP_BUFFER  "STATE This holds the state during an overlap so the next state can be determined" %
%   N9:13  PROC_OVERLAP  "STATE Process Purify Overlap" %
% Rung: 6 %
% TITLE: REGEN A %
% Entering SYSTEM STANDBY
% If the state of this machine is PURIFY B and the state of the system is STANDBY, then buffer the current state of this machine and go to the PROCESS STANDBY state %
SOR EQU N11:0 N9:12 EQU N10:0 N9:0 BST MOV N9:12 N11:3 NXB MOV N9:10 N11:0 BND EOR
%   N11:0  PROC_STATE  "STATE The current state of the process" %
%   N9:12  PROC_REGEN_A  "STATE Process Purify B" %
%   N10:0  SYSTEM_STATE  "<datalog> The current state of the system" %
%   N9:0  SYSTEM_STANDBY  "STATE System Standby" %
%   N11:3  PROC_STANDBY_BUFFER  "STATE This holds the state of the machine when the system enters STANDBY state" %
%   N9:10  PROCESS_STANDBY %

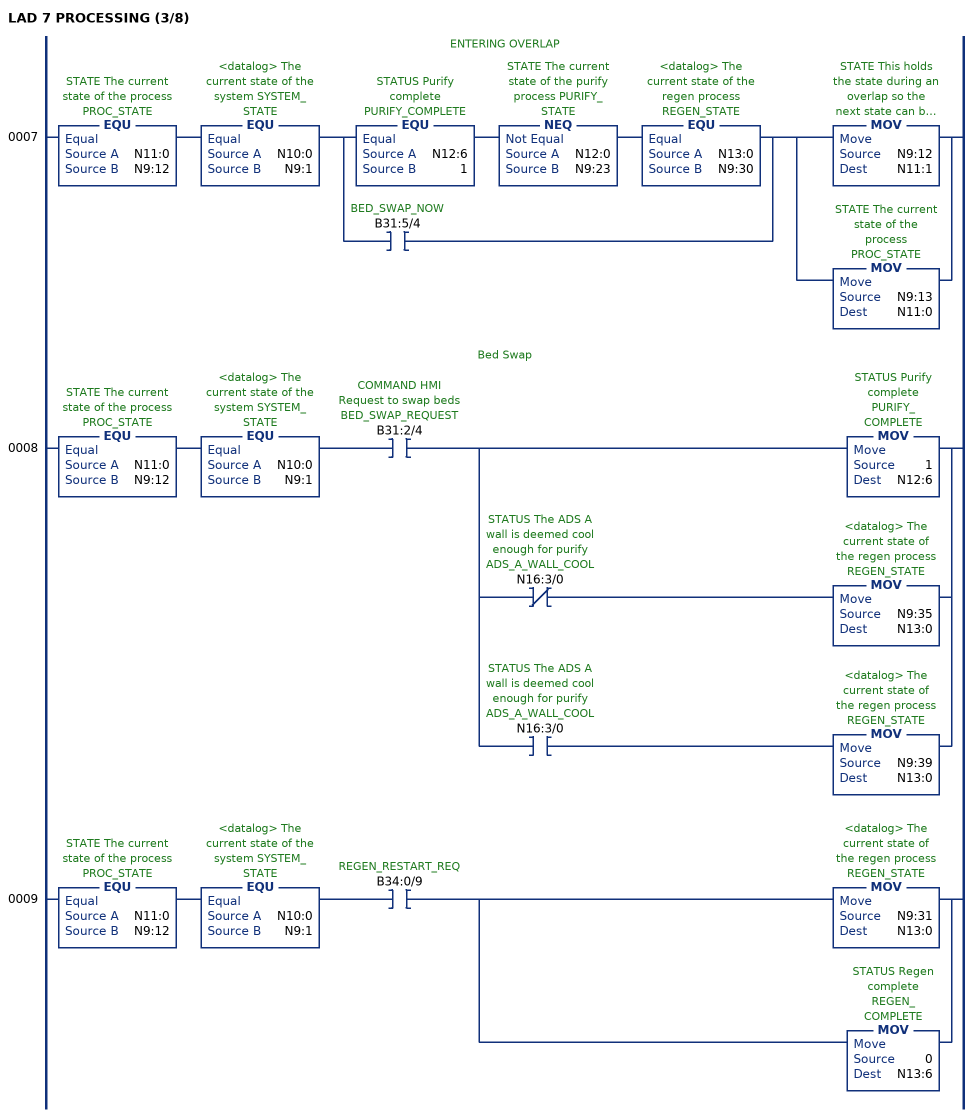
% Rung: 7 %
% ENTERING OVERLAP %
SOR EQU N11:0 N9:12 EQU N10:0 N9:1 BST EQU N12:6 1 NEQ N12:0 N9:23 EQU N13:0 N9:30 NXB XIC B31:5/4 BND BST MOV N9:12 N11:1 NXB MOV N9:13 N11:0 BND EOR
%   N11:0  PROC_STATE  "STATE The current state of the process" %
%   N9:12  PROC_REGEN_A  "STATE Process Purify B" %
%   N10:0  SYSTEM_STATE  "<datalog> The current state of the system" %
%   N9:1  SYSTEM_PROCESS  "STATE System Process" %
%   N12:6  PURIFY_COMPLETE  "STATUS Purify complete" %
%   N12:0  PURIFY_STATE  "STATE The current state of the purify process" %
%   N9:23  PURIFY_MANUAL_HOLD  "STATE Purify Manual Hold" %
%   N13:0  REGEN_STATE  "<datalog> The current state of the regen process" %
%   N9:30  REGEN_STANDBY  "STATE Regen Standby" %
%   B31:5/4  BED_SWAP_NOW %
%   N11:1  PROC_OVERLAP_BUFFER  "STATE This holds the state during an overlap so the next state can be determined" %
%   N9:13  PROC_OVERLAP  "STATE Process Purify Overlap" %
% Rung: 8 %
% Bed Swap %
SOR EQU N11:0 N9:12 EQU N10:0 N9:1 XIC B31:2/4 BST MOV 1 N12:6 NXB XIO N16:3/0 MOV N9:35 N13:0 NXB XIC N16:3/0 MOV N9:39 N13:0 BND EOR
%   N11:0  PROC_STATE  "STATE The current state of the process" %
%   N9:12  PROC_REGEN_A  "STATE Process Purify B" %
%   N10:0  SYSTEM_STATE  "<datalog> The current state of the system" %
%   N9:1  SYSTEM_PROCESS  "STATE System Process" %
%   B31:2/4  BED_SWAP_REQUEST  "COMMAND HMI Request to swap beds" %
%   N12:6  PURIFY_COMPLETE  "STATUS Purify complete" %
%   N16:3/0  ADS_A_WALL_COOL  "STATUS The ADS A wall is deemed cool enough for purify" %
%   N9:35  REGEN_COOL_WALL  "STATE Regen Cool wall" %
%   N13:0  REGEN_STATE  "<datalog> The current state of the regen process" %
%   N9:39  REGEN_EQUALIZE %
% Rung: 9 %
SOR EQU N11:0 N9:12 EQU N10:0 N9:1 XIC B34:0/9 BST MOV N9:31 N13:0 NXB MOV 0 N13:6 BND EOR
%   N11:0  PROC_STATE  "STATE The current state of the process" %
%   N9:12  PROC_REGEN_A  "STATE Process Purify B" %
%   N10:0  SYSTEM_STATE  "<datalog> The current state of the system" %
%   N9:1  SYSTEM_PROCESS  "STATE System Process" %
%   B34:0/9  REGEN_RESTART_REQ %
%   N9:31  REGEN_DELAY  "STATE Regen Delay" %
%   N13:0  REGEN_STATE  "<datalog> The current state of the regen process" %
%   N13:6  REGEN_COMPLETE  "STATUS Regen complete" %

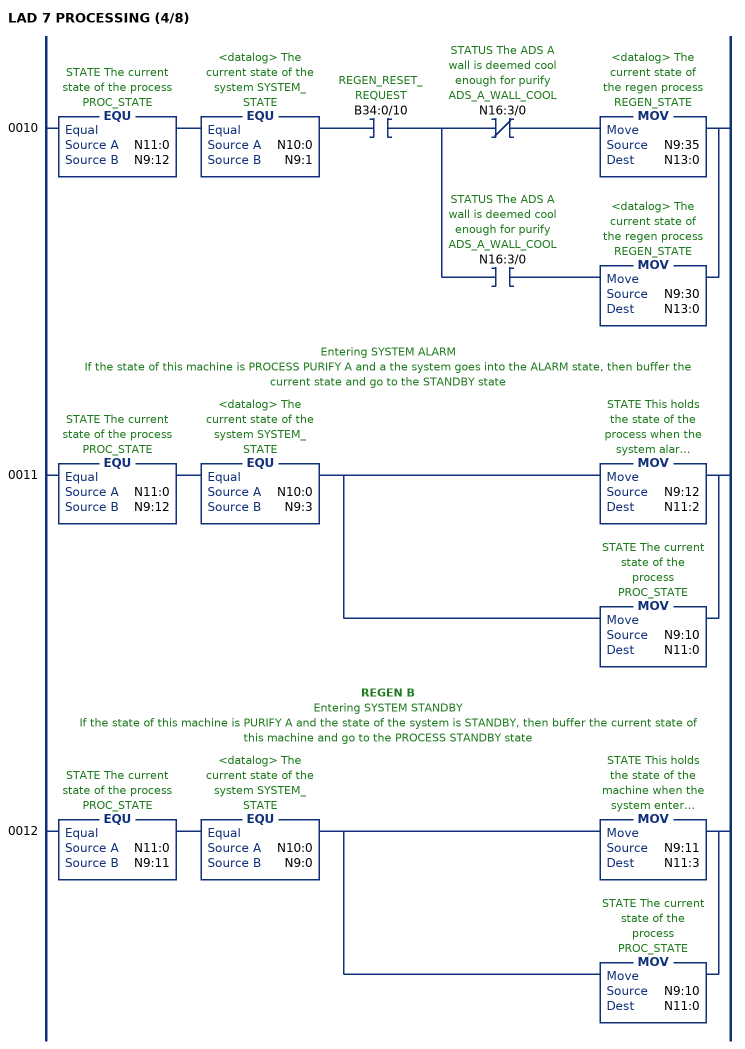
% Rung: 10 %
SOR EQU N11:0 N9:12 EQU N10:0 N9:1 XIC B34:0/10 BST XIO N16:3/0 MOV N9:35 N13:0 NXB XIC N16:3/0 MOV N9:30 N13:0 BND EOR
%   N11:0  PROC_STATE  "STATE The current state of the process" %
%   N9:12  PROC_REGEN_A  "STATE Process Purify B" %
%   N10:0  SYSTEM_STATE  "<datalog> The current state of the system" %
%   N9:1  SYSTEM_PROCESS  "STATE System Process" %
%   B34:0/10  REGEN_RESET_REQUEST %
%   N16:3/0  ADS_A_WALL_COOL  "STATUS The ADS A wall is deemed cool enough for purify" %
%   N9:35  REGEN_COOL_WALL  "STATE Regen Cool wall" %
%   N13:0  REGEN_STATE  "<datalog> The current state of the regen process" %
%   N9:30  REGEN_STANDBY  "STATE Regen Standby" %
% Rung: 11 %
% Entering SYSTEM ALARM
% If the state of this machine is PROCESS PURIFY A and a the system goes into the ALARM state, then buffer the current state and go to the STANDBY state %
SOR EQU N11:0 N9:12 EQU N10:0 N9:3 BST MOV N9:12 N11:2 NXB MOV N9:10 N11:0 BND EOR
%   N11:0  PROC_STATE  "STATE The current state of the process" %
%   N9:12  PROC_REGEN_A  "STATE Process Purify B" %
%   N10:0  SYSTEM_STATE  "<datalog> The current state of the system" %
%   N9:3  SYSTEM_ALARM  "STATE System Alarm" %
%   N11:2  PROC_ALARM_BUFFER  "STATE This holds the state of the process when the system alarm occured" %
%   N9:10  PROCESS_STANDBY %
% Rung: 12 %
% TITLE: REGEN B %
% Entering SYSTEM STANDBY
% If the state of this machine is PURIFY A and the state of the system is STANDBY, then buffer the current state of this machine and go to the PROCESS STANDBY state %
SOR EQU N11:0 N9:11 EQU N10:0 N9:0 BST MOV N9:11 N11:3 NXB MOV N9:10 N11:0 BND EOR
%   N11:0  PROC_STATE  "STATE The current state of the process" %
%   N9:11  PROC_REGEN_B  "STATE Process Purify A" %
%   N10:0  SYSTEM_STATE  "<datalog> The current state of the system" %
%   N9:0  SYSTEM_STANDBY  "STATE System Standby" %
%   N11:3  PROC_STANDBY_BUFFER  "STATE This holds the state of the machine when the system enters STANDBY state" %
%   N9:10  PROCESS_STANDBY %

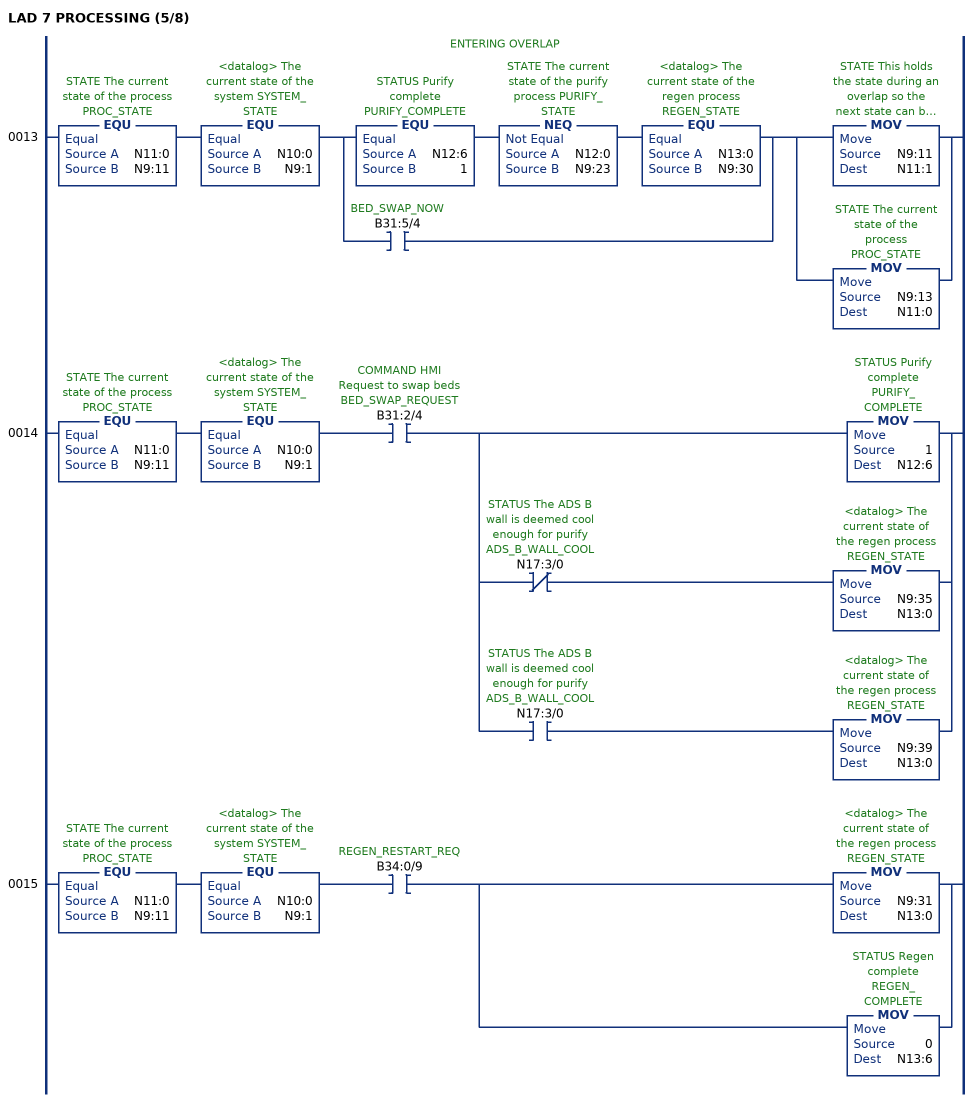
% Rung: 13 %
% ENTERING OVERLAP %
SOR EQU N11:0 N9:11 EQU N10:0 N9:1 BST EQU N12:6 1 NEQ N12:0 N9:23 EQU N13:0 N9:30 NXB XIC B31:5/4 BND BST MOV N9:11 N11:1 NXB MOV N9:13 N11:0 BND EOR
%   N11:0  PROC_STATE  "STATE The current state of the process" %
%   N9:11  PROC_REGEN_B  "STATE Process Purify A" %
%   N10:0  SYSTEM_STATE  "<datalog> The current state of the system" %
%   N9:1  SYSTEM_PROCESS  "STATE System Process" %
%   N12:6  PURIFY_COMPLETE  "STATUS Purify complete" %
%   N12:0  PURIFY_STATE  "STATE The current state of the purify process" %
%   N9:23  PURIFY_MANUAL_HOLD  "STATE Purify Manual Hold" %
%   N13:0  REGEN_STATE  "<datalog> The current state of the regen process" %
%   N9:30  REGEN_STANDBY  "STATE Regen Standby" %
%   B31:5/4  BED_SWAP_NOW %
%   N11:1  PROC_OVERLAP_BUFFER  "STATE This holds the state during an overlap so the next state can be determined" %
%   N9:13  PROC_OVERLAP  "STATE Process Purify Overlap" %
% Rung: 14 %
SOR EQU N11:0 N9:11 EQU N10:0 N9:1 XIC B31:2/4 BST MOV 1 N12:6 NXB XIO N17:3/0 MOV N9:35 N13:0 NXB XIC N17:3/0 MOV N9:39 N13:0 BND EOR
%   N11:0  PROC_STATE  "STATE The current state of the process" %
%   N9:11  PROC_REGEN_B  "STATE Process Purify A" %
%   N10:0  SYSTEM_STATE  "<datalog> The current state of the system" %
%   N9:1  SYSTEM_PROCESS  "STATE System Process" %
%   B31:2/4  BED_SWAP_REQUEST  "COMMAND HMI Request to swap beds" %
%   N12:6  PURIFY_COMPLETE  "STATUS Purify complete" %
%   N17:3/0  ADS_B_WALL_COOL  "STATUS The ADS B wall is deemed cool enough for purify" %
%   N9:35  REGEN_COOL_WALL  "STATE Regen Cool wall" %
%   N13:0  REGEN_STATE  "<datalog> The current state of the regen process" %
%   N9:39  REGEN_EQUALIZE %
% Rung: 15 %
SOR EQU N11:0 N9:11 EQU N10:0 N9:1 XIC B34:0/9 BST MOV N9:31 N13:0 NXB MOV 0 N13:6 BND EOR
%   N11:0  PROC_STATE  "STATE The current state of the process" %
%   N9:11  PROC_REGEN_B  "STATE Process Purify A" %
%   N10:0  SYSTEM_STATE  "<datalog> The current state of the system" %
%   N9:1  SYSTEM_PROCESS  "STATE System Process" %
%   B34:0/9  REGEN_RESTART_REQ %
%   N9:31  REGEN_DELAY  "STATE Regen Delay" %
%   N13:0  REGEN_STATE  "<datalog> The current state of the regen process" %
%   N13:6  REGEN_COMPLETE  "STATUS Regen complete" %

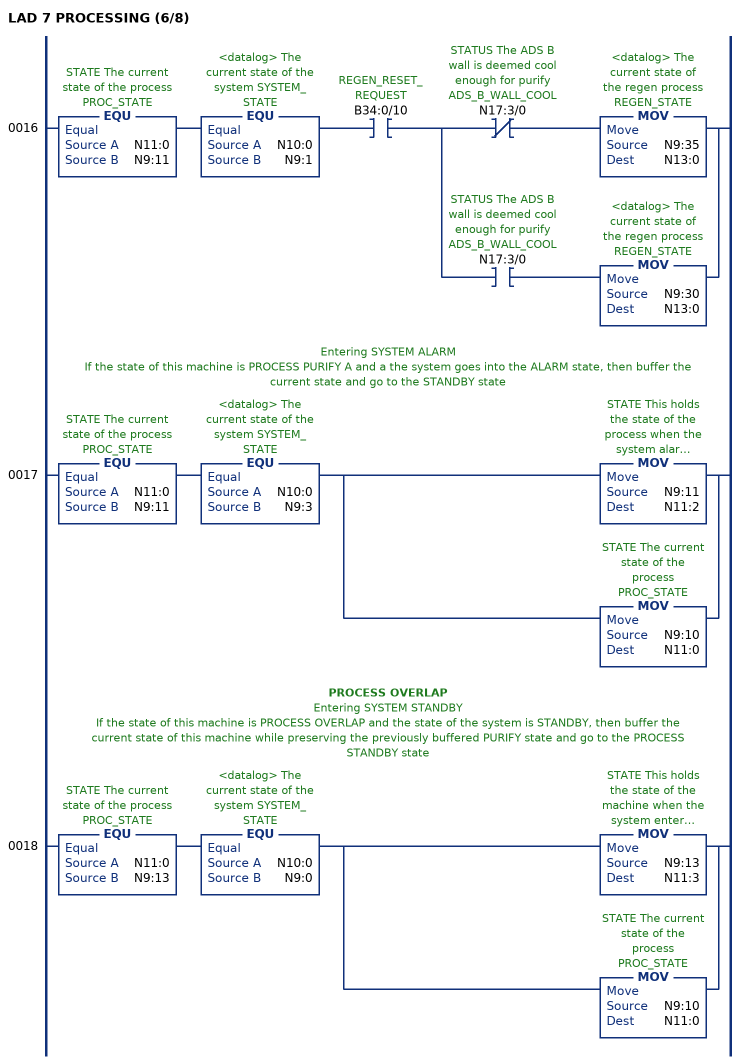
% Rung: 16 %
SOR EQU N11:0 N9:11 EQU N10:0 N9:1 XIC B34:0/10 BST XIO N17:3/0 MOV N9:35 N13:0 NXB XIC N17:3/0 MOV N9:30 N13:0 BND EOR
%   N11:0  PROC_STATE  "STATE The current state of the process" %
%   N9:11  PROC_REGEN_B  "STATE Process Purify A" %
%   N10:0  SYSTEM_STATE  "<datalog> The current state of the system" %
%   N9:1  SYSTEM_PROCESS  "STATE System Process" %
%   B34:0/10  REGEN_RESET_REQUEST %
%   N17:3/0  ADS_B_WALL_COOL  "STATUS The ADS B wall is deemed cool enough for purify" %
%   N9:35  REGEN_COOL_WALL  "STATE Regen Cool wall" %
%   N13:0  REGEN_STATE  "<datalog> The current state of the regen process" %
%   N9:30  REGEN_STANDBY  "STATE Regen Standby" %
% Rung: 17 %
% Entering SYSTEM ALARM
% If the state of this machine is PROCESS PURIFY A and a the system goes into the ALARM state, then buffer the current state and go to the STANDBY state %
SOR EQU N11:0 N9:11 EQU N10:0 N9:3 BST MOV N9:11 N11:2 NXB MOV N9:10 N11:0 BND EOR
%   N11:0  PROC_STATE  "STATE The current state of the process" %
%   N9:11  PROC_REGEN_B  "STATE Process Purify A" %
%   N10:0  SYSTEM_STATE  "<datalog> The current state of the system" %
%   N9:3  SYSTEM_ALARM  "STATE System Alarm" %
%   N11:2  PROC_ALARM_BUFFER  "STATE This holds the state of the process when the system alarm occured" %
%   N9:10  PROCESS_STANDBY %
% Rung: 18 %
% TITLE: PROCESS OVERLAP %
% Entering SYSTEM STANDBY
% If the state of this machine is PROCESS OVERLAP and the state of the system is STANDBY, then buffer the current state of this machine while preserving the previously buffered PURIFY state and go to the PROCESS STANDBY state %
SOR EQU N11:0 N9:13 EQU N10:0 N9:0 BST MOV N9:13 N11:3 NXB MOV N9:10 N11:0 BND EOR
%   N11:0  PROC_STATE  "STATE The current state of the process" %
%   N9:13  PROC_OVERLAP  "STATE Process Purify Overlap" %
%   N10:0  SYSTEM_STATE  "<datalog> The current state of the system" %
%   N9:0  SYSTEM_STANDBY  "STATE System Standby" %
%   N11:3  PROC_STANDBY_BUFFER  "STATE This holds the state of the machine when the system enters STANDBY state" %
%   N9:10  PROCESS_STANDBY %

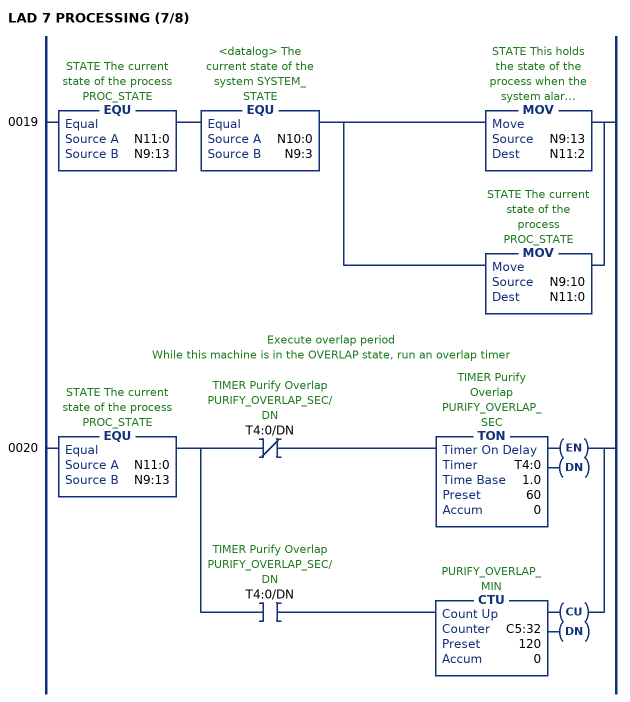
% Rung: 19 %
SOR EQU N11:0 N9:13 EQU N10:0 N9:3 BST MOV N9:13 N11:2 NXB MOV N9:10 N11:0 BND EOR
%   N11:0  PROC_STATE  "STATE The current state of the process" %
%   N9:13  PROC_OVERLAP  "STATE Process Purify Overlap" %
%   N10:0  SYSTEM_STATE  "<datalog> The current state of the system" %
%   N9:3  SYSTEM_ALARM  "STATE System Alarm" %
%   N11:2  PROC_ALARM_BUFFER  "STATE This holds the state of the process when the system alarm occured" %
%   N9:10  PROCESS_STANDBY %
% Rung: 20 %
% Execute overlap period
% While this machine is in the OVERLAP state, run an overlap timer %
SOR EQU N11:0 N9:13 BST XIO T4:0/DN TON T4:0 1.0 60 0 NXB XIC T4:0/DN CTU C5:32 120 0 BND EOR
%   N11:0  PROC_STATE  "STATE The current state of the process" %
%   N9:13  PROC_OVERLAP  "STATE Process Purify Overlap" %
%   T4:0  PURIFY_OVERLAP_SEC  "TIMER Purify Overlap" %
%   C5:32  PURIFY_OVERLAP_MIN %

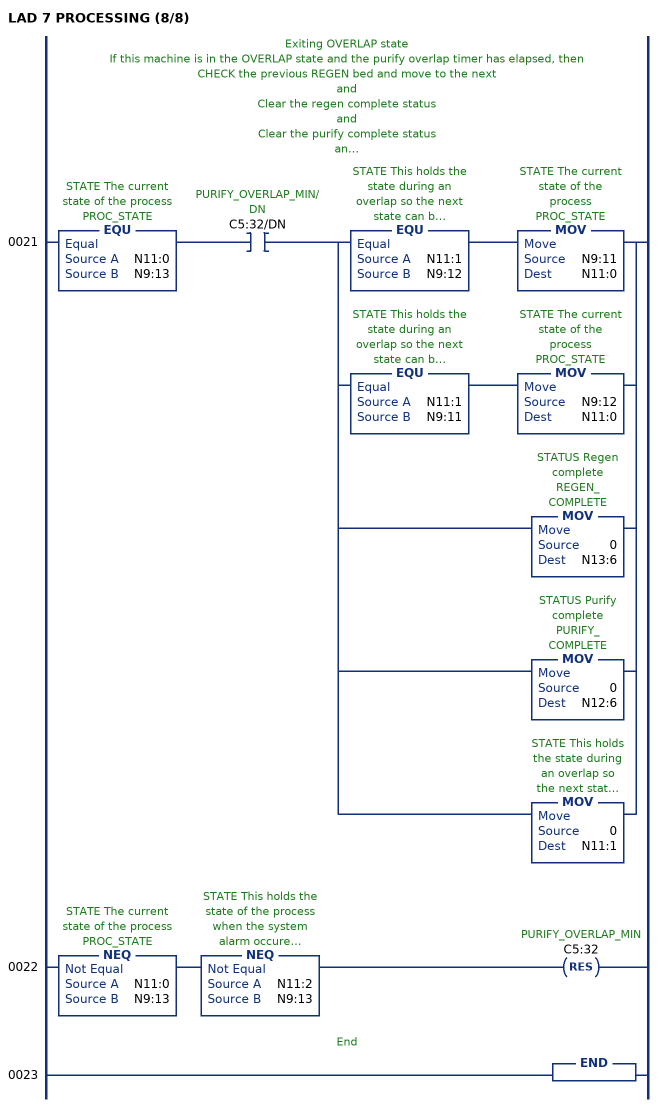
% Rung: 21 %
% Exiting OVERLAP state
% If this machine is in the OVERLAP state and the purify overlap timer has elapsed, then
% CHECK the previous REGEN bed and move to the next
% and
% Clear the regen complete status
% and
% Clear the purify complete status
% and
% clear the process buffer %
SOR EQU N11:0 N9:13 XIC C5:32/DN BST EQU N11:1 N9:12 MOV N9:11 N11:0 NXB EQU N11:1 N9:11 MOV N9:12 N11:0 NXB MOV 0 N13:6 NXB MOV 0 N12:6 NXB MOV 0 N11:1 BND EOR
%   N11:0  PROC_STATE  "STATE The current state of the process" %
%   N9:13  PROC_OVERLAP  "STATE Process Purify Overlap" %
%   C5:32  PURIFY_OVERLAP_MIN %
%   N11:1  PROC_OVERLAP_BUFFER  "STATE This holds the state during an overlap so the next state can be determined" %
%   N9:12  PROC_REGEN_A  "STATE Process Purify B" %
%   N9:11  PROC_REGEN_B  "STATE Process Purify A" %
%   N13:6  REGEN_COMPLETE  "STATUS Regen complete" %
%   N12:6  PURIFY_COMPLETE  "STATUS Purify complete" %
% Rung: 22 %
SOR NEQ N11:0 N9:13 NEQ N11:2 N9:13 RES C5:32 EOR
%   N11:0  PROC_STATE  "STATE The current state of the process" %
%   N9:13  PROC_OVERLAP  "STATE Process Purify Overlap" %
%   N11:2  PROC_ALARM_BUFFER  "STATE This holds the state of the process when the system alarm occured" %
%   C5:32  PURIFY_OVERLAP_MIN %
% Rung: 23 %
% End %
SOR END EOR

LADDER 8 "MANUAL_CTL"    % Runs the manual valve control %
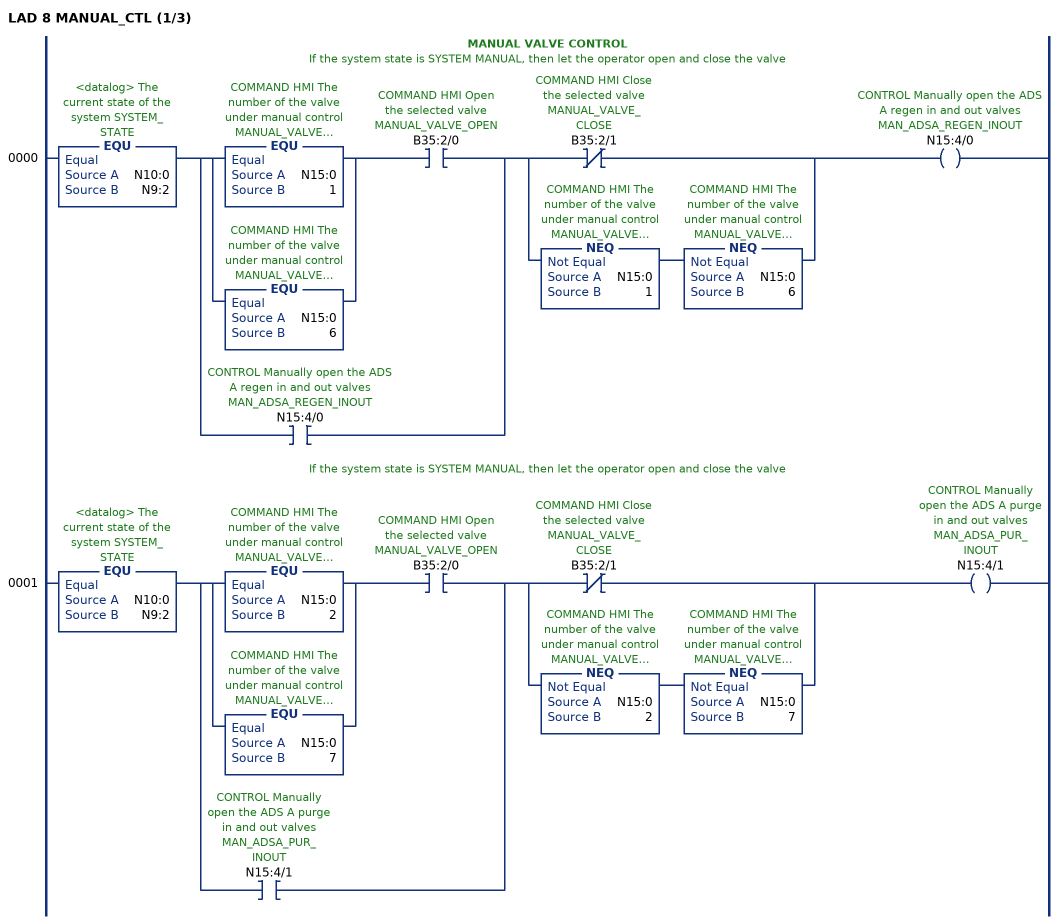
% Rung: 0 %
% TITLE: MANUAL VALVE CONTROL %
% If the system state is SYSTEM MANUAL, then let the operator open and close the valve %
SOR EQU N10:0 N9:2 BST BST EQU N15:0 1 NXB EQU N15:0 6 BND XIC B35:2/0 NXB XIC N15:4/0 BND BST XIO B35:2/1 NXB NEQ N15:0 1 NEQ N15:0 6 BND OTE N15:4/0 EOR
%   N10:0  SYSTEM_STATE  "<datalog> The current state of the system" %
%   N9:2  SYSTEM_MANUAL  "STATE System Manual" %
%   N15:0  MANUAL_VALVE_NUMBER  "COMMAND HMI The number of the valve under manual control" %
%   B35:2/0  MANUAL_VALVE_OPEN  "COMMAND HMI Open the selected valve" %
%   N15:4/0  MAN_ADSA_REGEN_INOUT  "CONTROL Manually open the ADS A regen in and out valves" %
%   B35:2/1  MANUAL_VALVE_CLOSE  "COMMAND HMI Close the selected valve" %
% Rung: 1 %
% If the system state is SYSTEM MANUAL, then let the operator open and close the valve %
SOR EQU N10:0 N9:2 BST BST EQU N15:0 2 NXB EQU N15:0 7 BND XIC B35:2/0 NXB XIC N15:4/1 BND BST XIO B35:2/1 NXB NEQ N15:0 2 NEQ N15:0 7 BND OTE N15:4/1 EOR
%   N10:0  SYSTEM_STATE  "<datalog> The current state of the system" %
%   N9:2  SYSTEM_MANUAL  "STATE System Manual" %
%   N15:0  MANUAL_VALVE_NUMBER  "COMMAND HMI The number of the valve under manual control" %
%   B35:2/0  MANUAL_VALVE_OPEN  "COMMAND HMI Open the selected valve" %
%   N15:4/1  MAN_ADSA_PUR_INOUT  "CONTROL Manually open the ADS A purge in and out valves" %
%   B35:2/1  MANUAL_VALVE_CLOSE  "COMMAND HMI Close the selected valve" %

